# B&R Automation Studio project PLC code - cp (part 10)

#### PressureCtrl.st
```iecst
ACTION PressureCtrl:

	//Send the data from the configuration to the PID structure
	LoadPIDparam(ADR(pidParPressure), ADR(dataVacc.Parameters.parPID));

	xEnablePID := StatusCtrl=TRANSVAC_WAITING OR StatusCtrl=TRANSVAC_CONTROLLING;

	//**********************************************************************************
	// PID PID PID PID PID PID PID PID PID PID PID PID PID PID PID PID PID PID PID PID
	//**********************************************************************************
	fbPIDPressure.Enable:=xEnablePID;
	fbPIDPressure.PIDParameters:=pidParPressure;
	fbPIDPressure.MinOut:=0.0;
	fbPIDPressure.MaxOut:= dataVacc.Parameters.rMaxPIDOut;
	fbPIDPressure.Update:= xUpdatePID;
	fbPIDPressure.EnableTracking := StatusCtrl=TRANSVAC_WAITING; //This is the manual mode
	fbPIDPressure.TrackingValue := dataVacc.Parameters.rStartUpDutyCycle; //The StartUp value is defined as Manual
	fbPIDPressure.SetValue:=dataVacc.Parameters.rVacPressureSetPointPerc;
	fbPIDPressure.ActValue:=rVacPressurePerc;
	fbPIDPressure();

	//Assignation of the SetPoint of the Blower
	CASE StatusCtrl OF

		TRANSVAC_OFF:
			dataVacc.Status.Blower.rDutyCycle:=0.0;

		TRANSVAC_WAITING,
		TRANSVAC_CONTROLLING:
			dataVacc.Status.Blower.rDutyCycle:=MAX(dataVacc.Parameters.rMinDutyCycle, fbPIDPressure.Out);

		TRANSVAC_MAN:
			dataVacc.Status.Blower.rDutyCycle:=MAX(dataVacc.Parameters.rMinDutyCycle, dataVacc.parSw.rManSetPoint);

	END_CASE

	ValveControl;

END_ACTION

ACTION ValveControl:

	IF StatusCtrl = TRANSVAC_OFF OR NOT dataVacc.Parameters.Hw.xSystemWithJoints THEN
		//When machine is in 0 all valves should be open --> no vacuum
		dataVacc.Outputs.VacuumValves := 0;
	ELSE
		//When working, open the valves received from Sw in the command. If a Mask of minimum vaccum is desired, applied here
		dataVacc.Outputs.VacuumValves := NOT (dataVacc.parSw.ValvMask OR dataVacc.Parameters.MinValvMask) ;
	END_IF

	//Set the status the same as the physical outputs
	dataVacc.Status.VacuumValves := dataVacc.Outputs.VacuumValves;

END_ACTION
```

#### BlowerAlarms.st
```iecst
ACTION BlowerAlarms:

	//Comunication Alarm
	IF Blower.Status.ErrorComms THEN
		dataVacc.Alarms.xAlrComsBlower := TRUE;
		dataVacc.Alarms.xAlrCommsBlower[uiIndex] := TRUE;
	END_IF

	tonCheckAlarms.IN := dataVacc.Inputs.xSafetyEnable;
	tonCheckAlarms.PT := T#3000ms;
	tonCheckAlarms();

	//Driver Blower Error
	IF tonCheckAlarms.Q AND NOT dataVacc.Alarms.xAlrComsBlower AND
		((Blower.Status.ErrorID <> 0 AND Blower.Status.ErrorID <> 20625) OR Blower.Status.StatusErrorStop) THEN
			dataVacc.Alarms.xAlrDriveBlowerError := TRUE;
			dataVacc.Alarms.xAlrBlowerError[uiIndex] := TRUE;
	END_IF

	//Separate CB Blower Alarm
	IF tonCheckAlarms.Q AND NOT Blower.ElecSignals.In.xBreakerOK THEN
		dataVacc.Alarms.xAlrBlowerCB[uiIndex] := TRUE;
	END_IF

	IF FALSE THEN
		dataVacc.Alarms.xAlrOvertorque := TRUE;
	END_IF

	//Alarm if the blower has a speed configure higher than 0, has order to move and is stopped
	//Using Orders.PowerOn because Commands.MovePositive and Commands.MoveNegative are just edges
	tonBlowerNotRunning[uiIndex].IN := StatusCtrl <> TRANSVAC_OFF AND Blower.Parameters.Velocity > 40.0 AND ABS(Blower.Status.ActVelocity) < 40.0;
	tonBlowerNotRunning[uiIndex].PT := T#5s;
	tonBlowerNotRunning[uiIndex]();
	IF tonBlowerNotRunning[uiIndex].Q THEN
		dataVacc.Alarms.xAlrBlowerNotRunning[uiIndex] := TRUE;
	END_IF

END_ACTION
```

#### BlowerControl.st
```iecst
ACTION BlowerControl:

	IF NOT Blower.Status.StatusOperation THEN
		xAllBlowersRunning := FALSE;
	END_IF

	IF NOT Blower.Status.xAtSpeed THEN
		xAllBlowersAtSpeed := FALSE;
	END_IF

	//Define maximum DutyCycle if in Maximum mode
	IF StatusCtrl = TRANSVAC_MAXIMUM THEN
		dataVacc.Status.Blower.rDutyCycle := 100;
	END_IF

	//TODO: Need to change units. Order from PID in % and command in rpm
	Blower.Parameters.Velocity := REAL_TO_UINT(dataVacc.Status.Blower.rDutyCycle * dataVacc.Parameters.rMaxSpeed / 100);

	xEnteringPowerOn := NOT dataVacc.Parameters.Mode.xZero AND NOT Blower.Orders.PowerOn;
	Blower.Orders.PowerOn := NOT dataVacc.Parameters.Mode.xZero;

	ConditionStart := Blower.Status.ReadyForOrders AND StatusCtrl <> TRANSVAC_OFF;

	IF ConditionStart AND NOT ConditionStart_copy  THEN
		//TOREVIEW: Command should be an edge
		IF BlowerDirection = MOTOR_POSITIVE THEN
			Blower.Commands.MovePositive := TRUE;
		ELSIF BlowerDirection = MOTOR_NEGATIVE THEN
			Blower.Commands.MoveNegative := TRUE;
		END_IF
	END_IF

	IF StatusCtrl = TRANSVAC_OFF AND StatusCtrl_copy<> TRANSVAC_OFF THEN
		Blower.Commands.Stop := TRUE;
	END_IF

	IF dataVacc.Commands.xReset OR xEnteringPowerOn THEN
		Blower.Commands.Reset := TRUE;
	END_IF

END_ACTION
```

#### EventLog.st
```iecst
ACTION LogStopAlarm:

	stEventLog.Source := ELOG_TYPE_TRANS_VACUUM;
	stEventLog.Severity:= ELOG_SEVERITY_INFO;
	stEventLog.Facility:= iIndexTransVacuum;
	stEventLog.ErrorCode:=0;

	stEventLog.Text := 'Vacuum.LogStopAlarm';

	IF 		iReasonStop.0 THEN stEventLog.Text := 'Vacuum. xAlrVacuumSensor';
	ELSIF 	iReasonStop.1 THEN stEventLog.Text := 'Vacuum. xAlrComsBlower';
	ELSIF 	iReasonStop.2 THEN stEventLog.Text := 'Vacuum. xAlrDriveBlowerError';
	ELSIF 	iReasonStop.3 THEN stEventLog.Text := 'Vacuum. xAlrOvertorque';
	ELSIF 	iReasonStop.4 THEN stEventLog.Text := 'Vacuum. xAlrJointSystemPressure';
	ELSIF 	iReasonStop.5 THEN stEventLog.Text := 'Vacuum. xAlrBlowersAnyCB';
	ELSIF 	iReasonStop.6 THEN stEventLog.Text := 'Vacuum. xAlrBlowerCB[1]';
	ELSIF 	iReasonStop.7 THEN stEventLog.Text := 'Vacuum. xAlrBlowerCB[2]';
	END_IF

	gEventLogLoader(EventData := ADR(stEventLog));

END_ACTION
```

### Program Logical/ExtPack/_Transport/TransVacuumCtrl/TransVacuumSim/TransVacuumSim_v1/TransVacuumSim (IEC)

#### Main.st
```iecst
PROGRAM _INIT
	pressureSim.AnalogType := ANALOGSIM_EXPONENTIAL_POS;
	pressureSim.rInitialValue := 16384;
	//pressureSim.rNewPresentValue := 16384;
	pressureSim.rMinValue := 10900;
	pressureSim.rMaxValue := 16384;

	rAParam := 5;	//Fixed change
	rBParam := 0.010;	//Change with DC

END_PROGRAM

PROGRAM _CYCLIC

	transVacc ACCESS ADR(gTransVacuum[iTransVacummSimIndex]);

	pressureSim.rA := rAParam * transVacc.Parameters.rMaxSystemVacuum;
	pressureSim.rB := rBParam * transVacc.Parameters.rMaxSystemVacuum;

	pressureSim.rActionControl := transVacc.Status.Blower.rDutyCycle;
	//pressureSim.xUseNewValue := EDGEPOS(transVacc.Status.State<>TRANSVAC_OFF);
	pressureSim();
	transVacc.Inputs.iPressureRaw:=REAL_TO_INT(pressureSim.rPresentValue);

	tofNoVacc.IN := transVacc.Status.rVacPressure > 0.0;
	tofNoVacc.PT := t#100ms;
	tofNoVacc();
	transVacc.Inputs.xJointSystemPressure	:= tofNoVacc.Q;
	transVacc.Inputs.xVaccAirFlow	:= tofNoVacc.Q;

	//Increase the index for simulating the next item
	iTransVacummSimIndex := iTransVacummSimIndex +1;

END_PROGRAM
```

### JamDetect.typ
```iecst
TYPE
	JamVibrationStatus_enum :
		(
		JAMVIB_NOT_INSTALLED,
		JAMVIB_NOT_INIT,
		JAMVIB_TESTING,
		JAMVIB_WORKING,
		JAMVIB_WAITING
		);
	JamTestingStatus_enum :
		(
		JAMVIBT_INIT,
		JAMVIBT_ACTIVATE_SIGNAL,
		JAMVIBT_WAITING_TO_CHECK,
		JAMVIBT_CHECKING,
		JAMVIBT_GO_NEXT
		);
	JamDetectInputs_typ : 	STRUCT
		xJamCrash : ARRAY[0..4]OF BOOL; (*Crash Bar Signal*)
		xJamTestOk : BOOL; (*Jam detection test has failed signal*)
		xJamLowCrash : BOOL; (*Low level crash device signal*)
	END_STRUCT;
	JamDetectOutputs_typ : 	STRUCT
		xJamTestSignal : ARRAY[0..4]OF BOOL; (*Jam test output signal*)
	END_STRUCT;
	JamDetectAlarms_typ : 	STRUCT
		xAlrJamCrash : ARRAY[0..4]OF BOOL; (*Alarm Stop, Crash in bar has detected*)
		xAlrJamTest : ARRAY[0..4]OF BOOL; (*Alarm Stop, Test has failed*)
		xAlrJamLowCrash : BOOL; (*Alarm Warning, low level crash detected in unknow bar*)
	END_STRUCT;
	JamDetectParameters_typ : 	STRUCT
		xJamEnabled : BOOL; (*Jam detection has enabled*)
		iMappingJam : INT; (*Physical mapping of the JamDevice*)
		iBlock : USINT; (*Block where the JamDevice is installed*)
		iMappingBarPos : ARRAY[0..MAX_LAST_JAMSENSOR]OF USINT; (*Physical Mapping Bar Position of the sensor*)
		xBarInstalled : ARRAY[0..MAX_LAST_JAMSENSOR]OF BOOL; (*Bar Installed*)
		iSensorsQuantity : USINT; (*Number of bars controlled by module*)
		xDisableTest : BOOL; (*Disables the JAMVIB_TESTING step*)
		iLowJamTimes : ARRAY[0..1]OF USINT; (*Number of rise edges of xJamLowCrash to show alarm*)
		iLowJamCheckDuration : ARRAY[0..1]OF TIME; (*Period of time to check consecutive xJamLowCrash rise edges to show alarm*)
		xDisableLowJamAlarm : BOOL; (*Low level jam detection alarm disabled*)
	END_STRUCT;
	JamDetectCommands_typ : 	STRUCT
		xReset : BOOL; (*Reset signal*)
		xMuteAlarms : BOOL; (*Mute alarms signal*)
		xStart : BOOL; (*Do the test and check*)
		xPause : BOOL; (*Jam pause comand, belt stop, bars in print and block in auto*)
	END_STRUCT;
	JamDetect_typ : 	STRUCT
		Inputs : JamDetectInputs_typ;
		Outputs : JamDetectOutputs_typ;
		Alarms : JamDetectAlarms_typ;
		Status : JamVibrationStatus_enum;
		Parameters : JamDetectParameters_typ;
		Commands : JamDetectCommands_typ;
		AlSummary : stEFI_AlarmSummary;
	END_STRUCT;
	JamPerBar_typ : 	STRUCT
		iJamDevice : USINT;
		iJamSensor : USINT;
		xAlrJamCrash : BOOL;
		xAlrJamTest : BOOL;
		xAlrLowJamCrash : BOOL; (*Low level jam detection from jam device*)
	END_STRUCT;
END_TYPE
```

### JamDetect.var
```iecst
VAR
	iIndexJam : USINT;
END_VAR
```

- Program Logical/ExtPack/_Transport/JamDetectCtrl/JamDetect_v1/InitJamDetect (IEC) (no source held here)

### Program Logical/ExtPack/_Transport/JamDetectCtrl/JamDetect_v1/JamDetect (IEC)

#### JamDetect.st - Init, cyclic, exit code
```iecst
PROGRAM _CYCLIC

	JamDetect ACCESS ADR(gJamDetect[iIndexJam]);

	IF NOT JamDetect.Parameters.xJamEnabled THEN
		JamDetect.Alarms := AlarmsReseted;
		JamDetect.Commands := CommandsReseted;

		JamDetect.Status := JAMVIB_NOT_INSTALLED;
		xTestFinished := FALSE;

		iIndexJam := iIndexJam + 1;
		RETURN;
	END_IF

	(***RESET ALARMS***)
	IF JamDetect.Commands.xReset THEN
		JamDetect.Alarms := AlarmsReseted;
		JamDetect.AlSummary.xAlarmStop := FALSE;
	END_IF

	JamDetectCtrl;
	JamAlarmsSound;

	iIndexJam := iIndexJam + 1;

END_PROGRAM
```

#### JamDetectCtrl.st - Chiller control
```iecst
ACTION JamDetectCtrl:

	xStatusChanged := StatusPrevious <> JamDetect.Status ;
	StatusPrevious := JamDetect.Status;

	CASE JamDetect.Status OF
		JAMVIB_NOT_INSTALLED:
			JamDetect.Status := JAMVIB_NOT_INIT;

		JAMVIB_NOT_INIT:
			ResetTestingOrders;
			IF JamDetect.Commands.xStart THEN
				IF JamDetect.Parameters.xDisableTest THEN
					JamDetect.Status := JAMVIB_WORKING;
				ELSIF NOT xAnyTestAlarm THEN
					JamDetect.Status := JAMVIB_TESTING;
				END_IF
			END_IF

		JAMVIB_TESTING:

			JamTesting;

			IF xTestFinished THEN
				IF JamDetect.Commands.xStart AND NOT xAnyTestAlarm THEN
					xTestFinished := FALSE;
					JamDetect.Status := JAMVIB_WORKING;
				ELSE
					JamDetect.Status := JAMVIB_NOT_INIT;
				END_IF
			END_IF

		JAMVIB_WORKING:

			JamAlarms;

			IF JamDetect.Commands.xPause THEN
				JamDetect.Status := JAMVIB_WAITING;
			END_IF

			IF NOT JamDetect.Commands.xStart THEN
				JamDetect.Status := JAMVIB_NOT_INIT;
			END_IF

		JAMVIB_WAITING:

			IF NOT JamDetect.Commands.xPause THEN
				IF JamDetect.Commands.xStart THEN
					JamDetect.Status := JAMVIB_WORKING;
				ELSE
					JamDetect.Status := JAMVIB_NOT_INIT;
				END_IF
			END_IF

	END_CASE

	//Saving state history
	IF JamDetect.Status<>StateHistory[0] THEN
		FOR iIndexHistory:=iHistoryLines TO 1 BY -1 DO
			StateHistory[iIndexHistory]:=StateHistory[iIndexHistory-1];
		END_FOR;
		StateHistory[0]:=JamDetect.Status;
	END_IF

	//Alarm Summary
	xAnyCrashAlarm	:= FALSE;
	IF JamDetect.Status <> JAMVIB_TESTING THEN xAnyTestAlarm := FALSE; END_IF

	FOR iIndexSensor:=1 TO JamDetect.Parameters.iSensorsQuantity BY 1 DO
		IF JamDetect.Alarms.xAlrJamCrash[iIndexSensor] THEN xAnyCrashAlarm := TRUE; END_IF
		IF JamDetect.Alarms.xAlrJamTest[iIndexSensor] THEN	xAnyTestAlarm := TRUE; END_IF
	END_FOR
	JamDetect.AlSummary.xAlarmStop := xAnyCrashAlarm OR xAnyTestAlarm;

	JamDetect.AlSummary.xAnyWarning := JamDetect.Alarms.xAlrJamLowCrash;

END_ACTION
```

#### JamAlarms.st - Chiller control
```iecst
ACTION JamAlarms:

	(**CRASH ALARMS**)
	FOR iIndexSensor:=1 TO JamDetect.Parameters.iSensorsQuantity BY 1 DO
		//Jam Alarms if Enabled
		IF JamDetect.Parameters.xBarInstalled[iIndexSensor] THEN
			IF NOT JamDetect.Inputs.xJamCrash[iIndexSensor] THEN JamDetect.Alarms.xAlrJamCrash[iIndexSensor] := TRUE; END_IF
		END_IF
	END_FOR

	(** Low jam detection DELOREAN-2694 **)
	IF NOT JamDetect.Parameters.xDisableLowJamAlarm THEN
		tofConsecutiveLowJamDetected[0].IN := JamDetect.Inputs.xJamLowCrash;
		tofConsecutiveLowJamDetected[0].PT := JamDetect.Parameters.iLowJamCheckDuration[0];
		tofConsecutiveLowJamDetected[0]();

		ctuConsecutiveLowJamDetected[0].CU := JamDetect.Inputs.xJamLowCrash AND tofConsecutiveLowJamDetected[0].Q;
		ctuConsecutiveLowJamDetected[0].PV := JamDetect.Parameters.iLowJamTimes[0];
		ctuConsecutiveLowJamDetected[0].RESET := NOT tofConsecutiveLowJamDetected[0].Q;
		ctuConsecutiveLowJamDetected[0]();

		tofConsecutiveLowJamDetected[1].IN := JamDetect.Inputs.xJamLowCrash;
		tofConsecutiveLowJamDetected[1].PT := JamDetect.Parameters.iLowJamCheckDuration[1];
		tofConsecutiveLowJamDetected[1]();

		ctuConsecutiveLowJamDetected[1].CU := JamDetect.Inputs.xJamLowCrash AND tofConsecutiveLowJamDetected[1].Q;
		ctuConsecutiveLowJamDetected[1].PV := JamDetect.Parameters.iLowJamTimes[1];
		ctuConsecutiveLowJamDetected[1].RESET := NOT tofConsecutiveLowJamDetected[1].Q;
		ctuConsecutiveLowJamDetected[1]();

		IF ctuConsecutiveLowJamDetected[0].Q OR ctuConsecutiveLowJamDetected[1].Q THEN
			JamDetect.Alarms.xAlrJamLowCrash := TRUE;
			LogWarningAlarm;
		END_IF
	END_IF

END_ACTION
```

#### JamAlarmsSound.st
```iecst
ACTION JamAlarmsSound:

	//Auto reset sound management. All alarms need to work with mute option
	ars_AlrJamDetectionSound(xAlarm:=JamDetect.AlSummary.xAlarmStop, xSilence:=JamDetect.Commands.xMuteAlarms);

	//AutoReset alarms.

		JamDetect.AlSummary.xAlarmSound:=ars_AlrJamDetectionSound.xAlarmSound;

END_ACTION
```

### Program Logical/ExtPack/_Transport/JamDetectCtrl/JamDetectSim/JamDetectSim_v1/JamDetectSim (IEC)

#### Main.st - Init, cyclic, exit code
```iecst
PROGRAM _CYCLIC
	(* Insert code here *)

	JamDetectData  ACCESS ADR(gJamDetect[usiJamDetectSimIndex]);
	JamDataSim ACCESS ADR(gSimJamDetect[usiJamDetectSimIndex]);

	IF NOT JamDetectData.Parameters.xJamEnabled THEN
		usiJamDetectSimIndex := usiJamDetectSimIndex +1;
		RETURN;
	END_IF

	JamDetectData.Inputs.xJamCrash[1]:=JamDetectData.Parameters.xBarInstalled[1] AND NOT JamDataSim.Commands.CreateCrash[1];
	JamDetectData.Inputs.xJamCrash[2]:=JamDetectData.Parameters.xBarInstalled[2] AND NOT JamDataSim.Commands.CreateCrash[2];
	JamDetectData.Inputs.xJamCrash[3]:=JamDetectData.Parameters.xBarInstalled[3] AND NOT JamDataSim.Commands.CreateCrash[3];
	JamDetectData.Inputs.xJamCrash[4]:=JamDetectData.Parameters.xBarInstalled[4] AND NOT JamDataSim.Commands.CreateCrash[4];

	//Tests

	tonTestDelay.IN :=	(JamDetectData.Outputs.xJamTestSignal[1]  AND NOT JamDataSim.Commands.ErrorInTest[1]) OR
						(JamDetectData.Outputs.xJamTestSignal[2]  AND NOT JamDataSim.Commands.ErrorInTest[2]) OR
						(JamDetectData.Outputs.xJamTestSignal[3]  AND NOT JamDataSim.Commands.ErrorInTest[3]) OR
						(JamDetectData.Outputs.xJamTestSignal[4]  AND NOT JamDataSim.Commands.ErrorInTest[4]);
	tonTestDelay.PT := T#1s;
	tonTestDelay();
	JamDetectData.Inputs.xJamTestOk := tonTestDelay.Q;

	usiJamDetectSimIndex := usiJamDetectSimIndex + 1;

END_PROGRAM
```

#### JamDetectSim.var - Local variables
```iecst
VAR
	JamDetectData : REFERENCE TO JamDetect_typ;
	JamDataSim : REFERENCE TO JamDetectSim_typ;
	usiIndexTest : USINT;
	tonTestDelay : TON;
END_VAR
```

### JamDetectSim.typ
```iecst
TYPE
	JamDetectCommandsSim_typ : 	STRUCT
		ErrorInTest : ARRAY[0..4]OF BOOL;
		CreateCrash : ARRAY[0..4]OF BOOL;
	END_STRUCT;
	JamDetectSim_typ : 	STRUCT
		Commands : JamDetectCommandsSim_typ;
	END_STRUCT;
END_TYPE
```

### JamDetectSimGen.var
```iecst
VAR
	usiJamDetectSimIndex : USINT;
END_VAR
```

### EdgeHoldDown.typ
```iecst
TYPE
	EdgeHoldDown_typ : 	STRUCT
		ordersSw : EdgeHoldDownOrdersSw; (*Orders from sw*)
		commandsSw : EdgeHoldDownCommandsSw; (*Commands gui*)
		commands : EdgeHoldDownCommands; (*Commands gui*)
		orders : EdgeHoldDownOrders;
		parameters : EdgeHoldDownParameters; (*Parameters gui*)
		parSw : EdgeHoldDownParametersSw;
		status : EdgeHoldDownStatus; (*States potocell system*)
		Alarms : EdgeHoldDownAlarms; (*Alarms*)
		AlSummary : stEFI_AlarmSummary; (*Alarms Summary*)
		inputs : EdgeHoldDownInputs;
		Hw : EdgeHoldDownParametersHw_typ;
	END_STRUCT;
	EdgeHoldDownCommands : 	STRUCT
		xErrorRst : BOOL;
		xMute : BOOL;
		xStop : BOOL;
		AutoMode : stEFI_MachineAutoModes;
		Mode : StGeneral_States_Mode;
	END_STRUCT;
	EdgeHoldDownOrdersSw : 	STRUCT
		xMoveForward : BOOL;
		xMoveBackward : BOOL;
		xMoveUp : BOOL;
		xMoveDown : BOOL;
	END_STRUCT;
	EdgeHoldDownCommandsSw : 	STRUCT
		xReference : BOOL;
	END_STRUCT;
	EdgeHoldDownOrders : 	STRUCT
		xResetPosition : BOOL; (*Order to move adjustment systems to resting position*)
		xAdjustToMedia : BOOL; (*Order to move adjustment system to working position*)
	END_STRUCT;
	EdgeHoldDownParametersSw : 	STRUCT
		rBarsOffset : REAL := 15; (*Offset desired between metal bands height and bars position (mm)*)
		iOverlap : INT := 10; (*Overlap between metal bands and media (mm)*)
		xEnable : BOOL;
	END_STRUCT;
	EdgeHoldDownParameters : 	STRUCT
		xInstalled : BOOL; (*This variable is activated when this functionality is intalled and ready to be enabled*)
		xEnableMovements : BOOL; (*Movements are enabled. Safe to move the adjustment systems and not damage the bars*)
		rDistanceMetalBandToSki : REAL := 20; (*Distance between ski and metal band*)
		rWidthSp : REAL; (*Metal bands width position setpoint*)
		rBarsOffset : REAL; (*Offset desired between metal bands and printing bars height*)
		rBarsHeighSp : REAL; (*Bars heigh setpoint*)
		rBlockPosition : REAL; (*Block over ehd system position*)
		iAdjustmentSystemsNumber : USINT; (*Number of adjustment systems used by the edge hold down. Adjust system is composed by two motors*)
	END_STRUCT;
	EdgeHoldDownStatus : 	STRUCT
		xInstalled : BOOL;
		xEnabled : BOOL;
		xReferencing : BOOL;
		xReferenced : BOOL;
		xInRestingPosition : BOOL;
		xAdjustedToMedia : BOOL;
		xMoving : BOOL;
		xReady : BOOL;
		xInPosition : BOOL;
		iSystemState : EdgeHoldDownState := EHD_STOPPED;
		EdgeHoldDownType : EdgeHoldDownType_enum;
		rSkiPosition : REAL;
		xGoingRestPosition : BOOL;
		xAdjusting : BOOL;
		rBlockPrePrintingPosition : REAL := 40; (*Distance between ski and metal band*)
	END_STRUCT;
	EdgeHoldDownAlarms : 	STRUCT
		xParametersOutOfRange : BOOL; (*Active when order to adjust media received and parameters are out of requirements*)
		xMovementsNotEnabled : BOOL; (*Active when order to adjust to media received when movements are not enabled*)
		xJam : BOOL; (*Jam sensor has detect media while ehd is adjusted to media*)
		xNotReferenced : BOOL; (*System not referenced*)
	END_STRUCT;
	EdgeHoldDownState :
		(
		EHD_STOPPED,
		EHD_MANUAL,
		EHD_IDLE,
		EHD_ERROR
		);
	EdgeHoldDownAutoState :
		(
		EHD_OUT_OF_AUTO,
		EHD_MOVEMENTS_NOT_ENABLED,
		EHD_READY,
		EHD_ADJUSTING_STEP_1,
		EHD_ADJUSTING_STEP_2,
		EHD_ADJUSTING_STEP_3,
		EHD_RESTING_STEP_1,
		EHD_RESTING_STEP_2,
		EHD_RESTING_STEP_3
		);
	EdgeHoldDownPositionStates :
		(
		UNDEFINED,
		HOMING,
		RESTING_POSITION,
		GOING_TO_WORKING_POSITION,
		WORKING_POSITION,
		GOING_TO_RESTING_POSITION
		);
	EdgeHoldDownOutputs : 	STRUCT
	END_STRUCT;
	EdgeHoldDownInputs : 	STRUCT
		xJam : BOOL;
	END_STRUCT;
	EdgeHoldDownType_enum :
		(
		EHDTY_UNDEFINED,
		EHDTY_V1,
		EHDTY_V2
		);
	EdgeHoldDownParametersHw_typ : 	STRUCT
		iMinBarsOffset : UINT := 10;
		iMaxBarsOffset : UINT := 15;
		iMinOverlap : INT := 8;
		iMaxOverlap : INT := 15;
		rMinWidthAdjustment : REAL := 424; (*Distance between sliders when inductive sensor for minimum position is active*)
		rMaxDistanceMetalBandToBelt : REAL := 60; (*Limited height where ehd can be moved vertically when postioned wider than belt's widht to avoid crash with 6l chassis*)
	END_STRUCT;
END_TYPE
```

- EdgeHoldDown.graphml (not shown)

### Program Logical/ExtPack/_Transport/EdgeHoldDown/EdgeHoldDown_v1/EdgeHoldDown (IEC)

#### EdgeHoldDown.st - Init, cyclic, exit code
```iecst
PROGRAM _INIT
	FOR iIndexHistory:=0 TO iHistoryLines DO
		StateHistory[iIndexHistory]:=EHD_STOPPED;
	END_FOR
END_PROGRAM

PROGRAM _CYCLIC

	//////////////////////////////
	////// ASSIGN LOCAL VARS //////
	//////////////////////////////

	//Main data assignation
	data ACCESS ADR (gEdgeHoldDown);
	AdjustmentSystem ACCESS ADR (gPairedMotors);

	data.status.xInstalled := data.parameters.xInstalled;

	IF EDGEPOS(data.parSw.xEnable) THEN
		data.status.xEnabled:=TRUE;

	//EHD may be disabled whether is positioned over the belt guide (Resting position)
	ELSIF ((NOT data.parSw.xEnable AND data.commands.Mode.xAuto) OR EDGEPOS(NOT data.parSw.xEnable)) AND data.status.xInRestingPosition THEN
		data.status.xEnabled := FALSE;
	END_IF

	Configuration;

	data.parameters.iAdjustmentSystemsNumber := LIMIT(1, data.parameters.iAdjustmentSystemsNumber, MAX_EHD_ADJUST_SYSTEMS);
	data.parameters.xEnableMovements := ((AdjustmentSystem[1].Motor[1].rPositionMotor + iSafetyOffset) < data.parameters.rBlockPosition); //Review how to set this condition when more than one block is installed

	IF NOT data.status.xInstalled OR NOT data.status.xEnabled THEN
		data.Alarms:= stAlarmsReseted;
		data.AlSummary := stEhdAlarmSummaryReseted;
		data.AlSummary.xAlarmSound:=FALSE;

		data.status.iSystemState:= EHD_STOPPED;
		data.status.xReferenced:=FALSE;
		ResetSwOrders;
		RETURN;
	END_IF

	//Reset alarms
	IF data.commands.xErrorRst THEN data.Alarms:= stAlarmsReseted; END_IF

	//States manager
	MachineState;

	//Alarms
	AlarmsSummary;

	///////////////////////
	//Alarm Sound
	AlarmSounds;

	//Resetting commands coming from sw
	data.commandsSw := ResetCommandsSw;

END_PROGRAM
```

#### AlarmsSummary.st - alarms summary
```iecst
ACTION AlarmsSummary:

	//////////////////////////
	////// RESET ALARMS //////
	//////////////////////////
	// Pending do commands gdata.commands.xReset
	IF data.commands.xErrorRst THEN
		data.Alarms := stAlarmsReseted;
		data.AlSummary := stEhdAlarmSummaryReseted;
	END_IF

	//Alarms
	IF data.status.xMoving AND NOT data.parameters.xEnableMovements THEN
		data.Alarms.xMovementsNotEnabled:=TRUE;
	END_IF

	IF data.status.xAdjustedToMedia AND data.inputs.xJam THEN
		data.Alarms.xJam:=TRUE;
	END_IF

	IF data.orders.xAdjustToMedia THEN
		IF ((AdjustmentSystem[1].parameters.rMechPositionMax + 2) < AdjustmentSystem[1].parameters.rPositionDesired) OR
			((AdjustmentSystem[1].parameters.rMechPositionMin - 2) > AdjustmentSystem[1].parameters.rPositionDesired) OR
			((AdjustmentSystem[2].parameters.rMechPositionMax + 2) < AdjustmentSystem[2].parameters.rPositionDesired) OR
			((AdjustmentSystem[2].parameters.rMechPositionMin - 2) > AdjustmentSystem[2].parameters.rPositionDesired) THEN

			data.Alarms.xParametersOutOfRange:=TRUE;
		END_IF
	END_IF

	//Alarms summary
	//Stop
	iReasonStop.0 := AdjustmentSystem[1].AlSummary.xAlarmStop;
	iReasonStop.1 := AdjustmentSystem[2].AlSummary.xAlarmStop;
	iReasonStop.2 := data.Alarms.xNotReferenced;
	iReasonStop.3 := data.Alarms.xParametersOutOfRange;

	data.AlSummary.xAlarmStop := iReasonStop > 0;
	IF EDGEPOS(data.AlSummary.xAlarmStop) THEN
		data.AlSummary.iReasonStop[0] := iReasonStop;
		LogStopAlarm;
	ELSIF EDGEPOS(NOT data.commands.AutoMode.xStop AND NOT data.AlSummary.xAlarmStop) THEN
		data.AlSummary.iReasonStop[0] := 0;
	END_IF

	//Critical
	iReasonCritical.0 := AdjustmentSystem[1].AlSummary.xAlarmCritical;
	iReasonCritical.1 := AdjustmentSystem[2].AlSummary.xAlarmCritical;
	iReasonCritical.2 := data.Alarms.xMovementsNotEnabled;
	iReasonCritical.3 := data.Alarms.xJam;

	data.AlSummary.xAlarmCritical := iReasonCritical > 0;
	IF EDGEPOS(data.AlSummary.xAlarmCritical) THEN
		data.AlSummary.iReasonCritical := iReasonCritical;
		LogCriticalAlarm;
	ELSIF EDGEPOS(data.commands.Mode.xAuto AND NOT data.AlSummary.xAlarmCritical) THEN
		data.AlSummary.iReasonCritical := 0;
	END_IF

	//Warning
	// It is just used for drive alarms
	iAnyWarning.0 := AdjustmentSystem[1].AlSummary.xAnyWarning;
	iAnyWarning.1 := AdjustmentSystem[2].AlSummary.xAnyWarning;

	data.AlSummary.xAnyWarning:= iAnyWarning > 0;
	IF EDGEPOS(data.AlSummary.xAnyWarning) THEN
		data.AlSummary.iReasonWarning := iAnyWarning;
		LogWarningAlarm;
	ELSIF EDGEPOS(NOT data.AlSummary.xAnyWarning) THEN
		data.AlSummary.iReasonWarning := 0;
	END_IF

END_ACTION
```

#### AlarmSounds.st
```iecst
ACTION AlarmSounds:

	// Alarms reseteable sound management.
	ars_AlrStop.xAlarm:= data.AlSummary.xAlarmStop;
	ars_AlrStop.xSilence:= data.commands.xMute;
	ars_AlrStop();

	ars_AlrCritical.xAlarm:= data.AlSummary.xAlarmCritical;
	ars_AlrCritical.xSilence:= data.commands.xMute;
	ars_AlrCritical();

	ars_AlrWarning.xAlarm:= data.AlSummary.xAnyWarning;
	ars_AlrWarning.xSilence:= data.commands.xMute;
	ars_AlrWarning();

	data.AlSummary.xAlarmSound:= //ars_AlrWarning.xAlarmSound OR
									ars_AlrStop.xAlarmSound OR
									ars_AlrCritical.xAlarmSound;

END_ACTION
```

#### EventLog.st
```iecst
ACTION LogWarningAlarm:

	stWarningAlarmsLog.Source := ELOG_TYPE_EHD;
	stWarningAlarmsLog.Severity:= ELOG_SEVERITY_INFO;
	stWarningAlarmsLog.Facility:= 0;
	stWarningAlarmsLog.ErrorCode:=0;

	stWarningAlarmsLog.Text := 'EHD.LogWarningAlarm';

	IF iReasonWarning.0 THEN stWarningAlarmsLog.Text := 'AdjustmentSystem[1].AlSummary.xAnyWarning';
	ELSIF iReasonWarning.1 THEN	stWarningAlarmsLog.Text := 'AdjustmentSystem[2].AlSummary.xAnyWarning';
	END_IF

	gEventLogLoader(EventData := ADR(stWarningAlarmsLog));

END_ACTION

ACTION LogStopAlarm:

	stStopAlarmsLog.Source := ELOG_TYPE_EHD;
	stStopAlarmsLog.Severity:= ELOG_SEVERITY_INFO;
	stStopAlarmsLog.Facility:= 0;
	stStopAlarmsLog.ErrorCode:=0;

	stStopAlarmsLog.Text := 'EHD.LogStopAlarm';

	IF iReasonStop.0 THEN stStopAlarmsLog.Text := 'AdjustmentSystem[1].AlSummary.xAlarmStop';
	ELSIF iReasonStop.1 THEN stStopAlarmsLog.Text := 'AdjustmentSystem[2].AlSummary.xAlarmStop';
	ELSIF iReasonStop.2 THEN stStopAlarmsLog.Text := 'data.Alarms.xNotReferenced';
	ELSIF iReasonStop.3 THEN stStopAlarmsLog.Text := 'data.Alarms.xParametersOutOfRange';
	END_IF

	gEventLogLoader(EventData := ADR(stStopAlarmsLog));

END_ACTION

ACTION LogCriticalAlarm:

	stCriticalAlarmsLog.Source := ELOG_TYPE_EHD;
	stCriticalAlarmsLog.Severity:= ELOG_SEVERITY_ERROR;
	stCriticalAlarmsLog.Facility:= 0;
	stCriticalAlarmsLog.ErrorCode:=0;

	stWarningAlarmsLog.Text := 'EHD.LogCriticalAlarm';

	IF iReasonCritical.0 THEN stWarningAlarmsLog.Text := 'AdjustmentSystem[1].AlSummary.xAlarmCritical';
	ELSIF iReasonCritical.1 THEN stWarningAlarmsLog.Text := 'AdjustmentSystem[2].AlSummary.xAlarmCritical';
	ELSIF iReasonCritical.2 THEN stWarningAlarmsLog.Text := 'data.Alarms.xMovementsNotEnabled';
	ELSIF iReasonCritical.3 THEN stWarningAlarmsLog.Text := 'data.Alarms.xJam';
	END_IF

	gEventLogLoader(EventData := ADR(stCriticalAlarmsLog));

END_ACTION
```

- Program Logical/ExtPack/_Transport/PairedIclaMotors/PairedIclaMotors_v1/InitPairedIclaMotors (IEC) (no source held here)

### Program Logical/ExtPack/_Transport/PairedIclaMotors/PairedIclaMotors_v1/PairedIclaMotors (IEC)

#### PairedIclaMotors.st - Init, cyclic, exit code
```iecst
PROGRAM _INIT
	FOR iIndexHistory:=0 TO iHistoryLines DO
		StateHistory[iIndexHistory]:=NOT_USED;
	END_FOR
END_PROGRAM

PROGRAM _CYCLIC

	//Main data assignation
	data ACCESS ADR (gPairedMotors[iIndexPairedIclaMotors]);
	IclaMaster ACCESS ADR (gIcla[gPairedMotors[iIndexPairedIclaMotors].parameters.IndexIclaMaster]);
	IclaGear ACCESS ADR (gIcla[gPairedMotors[iIndexPairedIclaMotors].parameters.IndexIclaGear]);

	IndexIclaMaster:=gPairedMotors[iIndexPairedIclaMotors].parameters.IndexIclaMaster;
	IndexIclaGear:=gPairedMotors[iIndexPairedIclaMotors].parameters.IndexIclaGear;

	//Review limits
	iNumIclaMotors := LIMIT(1, data.parameters.iNumIclaMotors, MAX_EHD_MOTORS_PER_ADJUST_SYS);
	rPositionDesired := LIMIT(data.parameters.rMechPositionMin, data.parameters.rPositionDesired, data.parameters.rMechPositionMax);

	data.status.xInstalled := data.parameters.xInstalled;
	IF data.status.xInstalled THEN
		//Motors data
		FOR iIndexIclaMotor:=1 TO iNumIclaMotors DO
			//Motor parameters
			dataToMotors;
			dataFromMotors;

			//Conversions
			IF data.parameters.xPositionSensorInstalled THEN
				Conversions;
			END_IF
		END_FOR
	END_IF

	data.status.xEnabled := data.parameters.xEnabled;
	IF NOT data.status.xEnabled THEN

		data.Alarms:= stAlarmsReseted;
		data.AlSummary := stAlarmSummaryReseted;
		data.AlSummary.xAlarmSound:=FALSE;

		data.status.xReferenced:=FALSE;
		ResetCommands;

		//Prepare for the next element
		iIndexPairedIclaMotors:= iIndexPairedIclaMotors +1;

		RETURN;
	END_IF

	IclaMotors[1]:=IclaMaster;
	IclaMotors[2]:=IclaGear;

	//Resetting commands
	IF data.commands.Mode.xZero THEN
		ResetCommands;
	END_IF

	//Motors state
	MotorsMachineState;

	// ALARMS
	AlarmsSummary;

	//Alarm Sound
	AlarmSounds;

	//Assigning motor data
	IclaMaster := IclaMotors[1];
	IclaGear := IclaMotors[2];

	//Prepare for the next element
	iIndexPairedIclaMotors:= iIndexPairedIclaMotors +1;

END_PROGRAM
```

#### MotorsMachineState.st - states control
```iecst
ACTION MotorsMachineState:

	xManualMovementEnabled := 	(iSystemState=MANUAL) OR
								(iSystemState=JOGGING) OR
								(iSystemState=HOMING_STEP_1) OR
								(iSystemState=HOMING_STEP_2) OR
								(iSystemState=HOMING_STEP_3);

	//Check motors are positioned in desired position
	IF (iSystemState=MANUAL) OR (iSystemState=JOGGING) THEN
		AssignJogOrders;
	END_IF
	CheckAnyManualMovement;
	CheckAnyManualOrder;

	CheckMotorStopped;
	//CheckMotorReferenced;
	CheckMotorReady;
	CheckMotorPositioned;

	CASE iSystemState OF

		NOT_INITIALIZED:
			ResetMotorsCommands;
			RemoveOrderMoveAbsolute;

			IF NOT xMotorStopped THEN
				SetStopOrder;
			ELSE
				CheckControllerReady;
				IF xControllerReady THEN
					iSystemState:=POWER_ON;
				END_IF
			END_IF

		POWER_ON:
			RemoveStopOrder;
			SetPowerOn;
			CheckPowerOn;
			IF xPoweredOn THEN
				//Go directly to wait homing process
				iSystemState:=POWERED;
			END_IF

		POWERED:
			IF xMotorReady THEN
				iSystemState := STANDSTILL;
			END_IF

		STANDSTILL:
			IF data.commands.Mode.xManual THEN
				iSystemState:=MANUAL;

			ELSIF data.commands.Mode.xAuto AND xMotorsReferenced AND data.parameters.xMovementsEnabled THEN
				iSystemState := AUTO;
			END_IF

		MANUAL:
			IF EDGEPOS(data.commands.xReference) THEN
				xMotorsReferenced := FALSE;
				iSystemState := HOMING_STEP_1;

			ELSIF xAnyManualMovement THEN
				iSystemState:=JOGGING;
			END_IF

		JOGGING:
			CheckMotorReady;
			IF NOT xAnyManualOrder THEN
				iSystemState := STANDSTILL;
			END_IF

		HOMING_STEP_1:
			//To home directly if both homing sensors are active
			CheckReferencePositionReached;
			IF xReferencePositionReached AND xMotorReady THEN
				iSystemState := HOMING_STEP_2;
			END_IF

		HOMING_STEP_2:
			//Execute home order
			SetHomeOrder;
			IF xMotorReady THEN
				iSystemState := HOMING_STEP_3;
			END_IF

		HOMING_STEP_3:
			CheckMotorReferenced;
			IF xMotorsReferenced THEN
				iSystemState := STANDSTILL;
			ELSE
				RemoveHomeOrder;
				iSystemState := HOMING_STEP_2;
			END_IF

		AUTO:
			RemoveStopOrder;
			IF xMotorReady THEN
				IF NOT xMotorsInPosition THEN
					SetOrderMoveAbsolute;
				END_IF
			ELSE
				iSystemState := NOT_INITIALIZED;
			END_IF

			IF data.status.xMoving THEN
				iSystemState := RUNNING;
			END_IF

		RUNNING:
			//If the movement is finished or the desired position has changed
			tonMotorStopped(IN:=xMotorStopped, PT:=T#500ms);
			IF xMotorsInPosition OR tonMotorStopped.Q OR data.commands.xStop THEN
				RemoveOrderMoveAbsolute;
				SetStopOrder;
				iSystemState := AUTO;
			END_IF

		ERROR:
			ResetMotorsCommands;
			//SetPowerOff;
			RemoveOrderMoveAbsolute;
			IF NOT xMotorStopped THEN
				SetStopOrder;
			END_IF

			IF NOT xAnyMotorError THEN
				iSystemState:=NOT_INITIALIZED;
			END_IF
	END_CASE

	//To check motors errors
	CheckAnyError;

	IF NOT data.parameters.xMovementsEnabled AND ((iSystemState = RUNNING) OR (iSystemState = AUTO)) THEN
		RemoveOrderMoveAbsolute;
		iSystemState := STANDSTILL;
	END_IF

	//Sending to ERROR
	IF xAnyMotorError OR data.AlSummary.xAlarmCritical THEN
		iSystemState:=ERROR;
	END_IF

	//In Zero mode it goes to not Init
	IF (data.commands.Mode.xZero) THEN
		iSystemState:=NOT_INITIALIZED;
	END_IF

	//Saving state history
	IF iSystemState<>StateHistory[0] THEN
		FOR iIndexHistory:=iHistoryLines TO 1 BY -1 DO
			StateHistory[iIndexHistory]:=StateHistory[iIndexHistory-1];
		END_FOR
		StateHistory[0]:=iSystemState;
	END_IF

	//State summary
	data.status.xInPosition := xMotorsInPosition;
	data.status.xMoving := NOT xMotorStopped;
	data.status.xReferenced	:= xMotorsReferenced;
	data.status.xReferencing :=	(iSystemState=HOMING_STEP_1) OR (iSystemState=HOMING_STEP_2) OR (iSystemState=HOMING_STEP_3);
	data.status.iSystemState := iSystemState;

END_ACTION

ACTION ResetMotorsCommands:
	FOR iIndexIclaMotor:=1 TO iNumIclaMotors DO
		IclaMotors[iIndexIclaMotor].Command.Enable := FALSE;
		IclaMotors[iIndexIclaMotor].Command.JogBackward := FALSE;
		IclaMotors[iIndexIclaMotor].Command.JogForward := FALSE;
		IclaMotors[iIndexIclaMotor].Command.MoveAbsolute := FALSE;
	END_FOR
END_ACTION

ACTION CheckControllerReady:
	xControllerReady:=TRUE;
	FOR iIndexIclaMotor:=1 TO iNumIclaMotors DO
		IF IclaMotors[iIndexIclaMotor].Status.Error.Communication THEN
			xControllerReady:=FALSE;
		END_IF
	END_FOR
END_ACTION

ACTION SetPowerOn:
	FOR iIndexIclaMotor:=1 TO iNumIclaMotors DO
		IclaMotors[iIndexIclaMotor].Command.Enable := TRUE;
	END_FOR
END_ACTION

ACTION SetPowerOff:
	FOR iIndexIclaMotor:=1 TO iNumIclaMotors DO
		IclaMotors[iIndexIclaMotor].Command.Enable := FALSE;
	END_FOR
END_ACTION

ACTION CheckPowerOn:
	xPoweredOn:=TRUE;
	FOR iIndexIclaMotor:=1 TO iNumIclaMotors DO
		IF (IclaMotors[iIndexIclaMotor].Status.IclaStatus<>AXISILE_POWER) AND (IclaMotors[iIndexIclaMotor].Status.IclaStatus<>AXISILE_READY) THEN
			xPoweredOn:=FALSE;
		END_IF
	END_FOR
END_ACTION

ACTION CheckMotorReady:
	xMotorReady:=TRUE;
	FOR iIndexIclaMotor:=1 TO iNumIclaMotors DO
		IF (IclaMotors[iIndexIclaMotor].Status.iDriveStatus<>ICLAST_ENABLE_OPERATION) THEN
			xMotorReady:=FALSE;
		END_IF
	END_FOR
END_ACTION

ACTION SetHomeOrder:
	FOR iIndexIclaMotor:=1 TO iNumIclaMotors DO
		IF IclaMotors[iIndexIclaMotor].Status.iActualVelocity = 0 THEN
			IclaMotors[iIndexIclaMotor].Command.Home := TRUE;
		END_IF
	END_FOR
END_ACTION

ACTION RemoveHomeOrder:
	FOR iIndexIclaMotor:=1 TO iNumIclaMotors DO
		IclaMotors[iIndexIclaMotor].Command.Home := FALSE;
	END_FOR
END_ACTION

ACTION SetOrderGoingForward:
	data.commands.xMoveForward := TRUE;
END_ACTION

ACTION RemoveOrderGoingForward:
	data.commands.xMoveForward := FALSE;
END_ACTION

ACTION SetOrderGoingBackward:
	data.commands.xMoveBackward := TRUE;
END_ACTION

ACTION RemoveOrderGoingBackward:
	data.commands.xMoveBackward := FALSE;
END_ACTION

ACTION SetOrderMoveAbsolute:
	rCopyPositionDesired := rPositionDesired;
	FOR iIndexIclaMotor:=1 TO iNumIclaMotors DO
		MotorDriveUnit.PositionDesired := data.Motor[iIndexIclaMotor].iDirection * rPositionDesired;
		MotorDriveUnit.Calculation := CALC_POS_PULSES;
		MotorDriveUnit();

		IclaMotors[iIndexIclaMotor].Parameter.MoveAbsolute.Position := REAL_TO_DINT(MotorDriveUnit.pulsesPositionDesired);
		IclaMotors[iIndexIclaMotor].Command.MoveAbsolute := TRUE;
	END_FOR
END_ACTION

ACTION RemoveOrderMoveAbsolute:
	FOR iIndexIclaMotor:=1 TO iNumIclaMotors DO
		IclaMotors[iIndexIclaMotor].Command.MoveAbsolute := FALSE;
	END_FOR
END_ACTION

ACTION SetStopOrder:
	FOR iIndexIclaMotor:=1 TO iNumIclaMotors DO
		IclaMotors[iIndexIclaMotor].Command.Stop := TRUE;
	END_FOR
END_ACTION

ACTION RemoveStopOrder:
	FOR iIndexIclaMotor:=1 TO iNumIclaMotors DO
		IclaMotors[iIndexIclaMotor].Command.Stop := FALSE;
	END_FOR
END_ACTION

ACTION AssignJogOrders:
	FOR iIndexIclaMotor:=1 TO iNumIclaMotors DO
		//[RGP] Ehd width fitting exit motor direction is not the same as the one on the entry side due to mechanical assembly.
		//This case does not apply to elevation motors, which are mechanically assembled the same way.
		IF iIndexPairedIclaMotors=2 AND iIndexIclaMotor=2 THEN
			IclaMotors[iIndexIclaMotor].Command.JogBackward := data.commands.xMoveForward AND NOT data.commands.xMoveBackward AND NOT data.Motor[iIndexIclaMotor].Inputs.xMinPositionReached;
			IclaMotors[iIndexIclaMotor].Command.JogForward := data.commands.xMoveBackward AND NOT data.commands.xMoveForward AND NOT data.Motor[iIndexIclaMotor].Inputs.xMaxPositionReached;
		ELSE
			IclaMotors[iIndexIclaMotor].Command.JogForward := data.commands.xMoveForward AND NOT data.commands.xMoveBackward AND NOT data.Motor[iIndexIclaMotor].Inputs.xMinPositionReached;
			IclaMotors[iIndexIclaMotor].Command.JogBackward := data.commands.xMoveBackward AND NOT data.commands.xMoveForward AND NOT data.Motor[iIndexIclaMotor].Inputs.xMaxPositionReached;
		END_IF
	END_FOR
END_ACTION

ACTION CheckAnyManualOrder:
	xAnyManualOrder := 	IclaMotors[1].Command.JogForward OR
						IclaMotors[1].Command.JogBackward OR
						IclaMotors[2].Command.JogForward OR
						IclaMotors[2].Command.JogBackward;
END_ACTION

ACTION CheckAnyManualMovement:
	xAnyManualMovement := FALSE;
	FOR iIndexIclaMotor:=1 TO iNumIclaMotors DO
		IF (IclaMotors[iIndexIclaMotor].Status.IclaStatus = AXISILE_JOG) THEN
			xAnyManualMovement := TRUE;
		END_IF
	END_FOR
END_ACTION

ACTION CheckAnyError:
	xAnyMotorError:=FALSE;
	FOR iIndexIclaMotor:=1 TO iNumIclaMotors DO
		// Not comms
		data.Motor[iIndexIclaMotor].Alarms.xCommsMotorError := FALSE;
		IF (IclaMotors[iIndexIclaMotor].Status.Error.Communication) THEN
			data.Motor[iIndexIclaMotor].Alarms.xCommsMotorError := TRUE;
		END_IF

		// Motor Error
		data.Motor[iIndexIclaMotor].Alarms.xMotorError := FALSE;
		IF ((IclaMotors[iIndexIclaMotor].Status.iDriveStatus = ICLAST_ERROR) OR
			IclaMotors[iIndexIclaMotor].Status.Error.ErrorNumber<>0) THEN
			data.Motor[iIndexIclaMotor].Alarms.xMotorError := TRUE;
		END_IF

		// Motor Error
		data.Motor[iIndexIclaMotor].Alarms.xControllerNotReady := FALSE;
		IF (IclaMotors[iIndexIclaMotor].Status.iDriveStatus = ICLAST_SWITCH_ON_DISABLED) THEN
			data.Motor[iIndexIclaMotor].Alarms.xControllerNotReady := TRUE;
		END_IF

	END_FOR
END_ACTION

ACTION CheckMotorStopped:
	xMotorStopped := TRUE;
	FOR iIndexIclaMotor:=1 TO iNumIclaMotors DO
		IF (IclaMotors[iIndexIclaMotor].Status.iActualVelocity <> 0) THEN
			xMotorStopped:=FALSE;
		END_IF
	END_FOR
END_ACTION

ACTION CheckReferencePositionReached:
	IF iIndexPairedIclaMotors=1 THEN
		//Elevation motors
		xReferencePositionReached := data.Motor[1].Inputs.xMinPositionReached AND data.Motor[2].Inputs.xMinPositionReached;
	ELSE
		//Width fitting motors
		xReferencePositionReached := data.Motor[1].Inputs.xMaxPositionReached AND data.Motor[2].Inputs.xMaxPositionReached;
	END_IF
END_ACTION

ACTION CheckMotorPositioned:
	xMotorsInPosition := TRUE;
	FOR iIndexIclaMotor:=1 TO iNumIclaMotors DO
		IF (ABS(data.Motor[iIndexIclaMotor].rPositionMotor - rPositionDesired) > data.Motor[iIndexIclaMotor].rMotorResolution) THEN
			xMotorsInPosition := FALSE;
		END_IF
	END_FOR
END_ACTION

ACTION CheckMotorReferenced:
	xMotorsReferenced := TRUE;
	FOR iIndexIclaMotor:=1 TO iNumIclaMotors DO
		IF NOT IclaMotors[iIndexIclaMotor].Status.xReferenced THEN
			xMotorsReferenced := FALSE;
		ELSE
			//Distance between sensors calculated instead of being a hardware defined parameter. Just for testing, this parameters must be defined by mechanical team
			data.Motor[iIndexIclaMotor].rDistanceBetweenSensors := (ABS(data.Motor[iIndexIclaMotor].rHomePosition)*2 + gEdgeHoldDown.Hw.rMinWidthAdjustment) - (data.Motor[iIndexIclaMotor].rMeasuredPositionFrontSide + data.Motor[iIndexIclaMotor].rMeasuredPositionBackSide);
		END_IF
	END_FOR
END_ACTION
```

#### Conversions.st
```iecst
ACTION Conversions:

	//There are two distance sensor per motor

	//y = mx + b
	//y = distance measured (mm)
	//x = value read by sensor
	//b = value of distance at minimum analogic value read (4mA) = 100mm
	//sensor maximum measure distance is 600

	//y(x)=0.0183x + 58 //Practical. (RawUnits)

	//Front sensor
	data.Motor[iIndexIclaMotor].rMeasuredPositionFrontSide := (data.Motor[iIndexIclaMotor].Inputs.iMeasuredPositionFrontSide*rSlopeAnalogSensor + rInterceptAnalogSensor);

	//Back sensor
	data.Motor[iIndexIclaMotor].rMeasuredPositionBackSide := (data.Motor[iIndexIclaMotor].Inputs.iMeasuredPositionBackSide*rSlopeAnalogSensor + rInterceptAnalogSensor);

	//Distance between metal bands/straps
	rMeasuredDistanceMetalStraps[iIndexIclaMotor] := 	data.Motor[iIndexIclaMotor].rMeasuredPositionFrontSide +
														data.Motor[iIndexIclaMotor].rMeasuredPositionBackSide +
														data.Motor[iIndexIclaMotor].rDistanceBetweenSensors;

	IF ABS(data.Motor[iIndexIclaMotor].rMeasuredDistanceMetalStraps - rMeasuredDistanceMetalStraps[iIndexIclaMotor])> rAnalogSensorTolerance THEN
		data.Motor[iIndexIclaMotor].rMeasuredDistanceMetalStraps := rMeasuredDistanceMetalStraps[iIndexIclaMotor];
	END_IF

END_ACTION
```

#### AlarmsSummary.st - alarms summary
```iecst
ACTION AlarmsSummary:

	//RESET ALARMS
	IF data.commands.xErrorRst THEN
		data.Alarms := stAlarmsReseted;
		data.AlSummary := stAlarmSummaryReseted;
	END_IF

	//Invalid position
	IF data.status.xReferenced AND data.status.xMoving THEN
		IF (rPositionMotorMm > (data.parameters.rMechPositionMax + data.Motor[1].rMotorResolution)) OR ((rPositionMotorMm < data.parameters.rMechPositionMin - data.Motor[1].rMotorResolution)) THEN
			data.Alarms.xPositionOutOfRange := TRUE;
		END_IF
	END_IF

	//Alarm Not referenced
	data.Alarms.xNotReferenced:= NOT data.status.xReferenced;

	//////////////////////////////////////////
	//To review in next releases how to share with SW an alarm per motor and not per adjustment system. To improve troubleshooting

	//Error general. Check error id for more information
	data.Alarms.xMotorError:=data.Motor[1].Alarms.xMotorError OR data.Motor[2].Alarms.xMotorError;

	//Enables (STO)
	IF data.Inputs.xSafetyEnable AND NOT data.commands.Mode.xZero THEN
		data.Alarms.xControllerNotReady :=  data.Motor[1].Alarms.xControllerNotReady OR data.Motor[2].Alarms.xControllerNotReady;
	END_IF

	//Comms
	data.Alarms.xCommsMotorError:=data.Motor[1].Alarms.xCommsMotorError OR data.Motor[2].Alarms.xCommsMotorError;

	xAnyMotorError := data.Alarms.xMotorError OR data.Alarms.xCommsMotorError;

	//////////////////////////////////////////

	//Motors not aligned
	data.Alarms.xNotAligned := ABS(data.Motor[1].rPositionMotor-data.Motor[2].rPositionMotor) > data.parameters.iMisalignmentTolerance;

	//Inconsistency between position measured (analogic input) and motor position information (motors encoder)
	iPositionMeasuredInconsistency.0 := ABS(data.Motor[1].rMetalStrapPos-data.Motor[1].rMeasuredDistanceMetalStraps) > data.parameters.iPositionResolution;
	iPositionMeasuredInconsistency.1 := ABS(data.Motor[2].rMetalStrapPos-data.Motor[2].rMeasuredDistanceMetalStraps) > data.parameters.iPositionResolution;

	IF iPositionMeasuredInconsistency>0 AND data.parameters.xPositionSensorInstalled AND xMotorStopped THEN
		data.Alarms.xPositionMeasuredInconsistency := TRUE;
	END_IF

	IF EDGEPOS(data.Alarms.xPositionMeasuredInconsistency) THEN
		rInputMeasuredDifference := (data.Motor[1].rMetalStrapPos-data.Motor[1].rMeasuredDistanceMetalStraps);
		rOutputMeasuredDifference := (data.Motor[2].rMetalStrapPos-data.Motor[2].rMeasuredDistanceMetalStraps);
	END_IF

	//Alarms summary
	//Stop
	iReasonStop.0 := data.Alarms.xMotorError;
	iReasonStop.1 := data.Alarms.xCommsMotorError;
	iReasonStop.2 := data.Alarms.xNotReferenced;
	iReasonStop.3 := xAnyMotorError;
	//iReasonStop.4 := data.Alarms.xPositionMeasuredInconsistency;

	data.AlSummary.xAlarmStop := iReasonStop > 0;
	IF EDGEPOS(data.AlSummary.xAlarmStop) THEN
		data.AlSummary.iReasonStop[0] := iReasonStop;
		LogStopAlarm;
	ELSIF EDGEPOS(NOT data.commands.AutoMode.xStop AND NOT data.AlSummary.xAlarmStop) THEN
		data.AlSummary.iReasonStop[0] := 0;
	END_IF

	//Critical
	iReasonCritical.0 := data.Alarms.xPositionOutOfRange;

	data.AlSummary.xAlarmCritical := iReasonCritical > 0;
	IF EDGEPOS(data.AlSummary.xAlarmCritical) THEN
		data.AlSummary.iReasonCritical := iReasonCritical;
		LogCriticalAlarm;
	ELSIF EDGEPOS(data.commands.Mode.xAuto AND NOT data.AlSummary.xAlarmCritical) THEN
		data.AlSummary.iReasonCritical := 0;
	END_IF

	//Warning
	// It is just used for drive alarms
	//iAnyWarning.0 := ;
	data.AlSummary.xAnyWarning:= iAnyWarning > 0;

	IF EDGEPOS(data.AlSummary.xAnyWarning) THEN
		data.AlSummary.iReasonWarning := iAnyWarning;
		LogWarningAlarm;
	ELSIF EDGEPOS(NOT data.AlSummary.xAnyWarning) THEN
		data.AlSummary.iReasonWarning := 0;
	END_IF

END_ACTION
```

#### AlarmSounds.st
```iecst
ACTION AlarmSounds:

	// Alarms reseteable sound management.
	ars_AlrStop.xAlarm:= data.AlSummary.xAlarmStop;
	ars_AlrStop.xSilence:= data.commands.xMute;
	ars_AlrStop();

	ars_AlrCritical.xAlarm:= data.AlSummary.xAlarmCritical;
	ars_AlrCritical.xSilence:= data.commands.xMute;
	ars_AlrCritical();

	ars_AlrWarning.xAlarm:= data.AlSummary.xAnyWarning;
	ars_AlrWarning.xSilence:= data.commands.xMute;
	ars_AlrWarning();

	data.AlSummary.xAlarmSound:= 	//ars_AlrWarning.xAlarmSound OR
									ars_AlrStop.xAlarmSound OR
									ars_AlrCritical.xAlarmSound OR
									(xAnyManualOrder AND gPLC.xBlk_200ms);

END_ACTION
```

#### ResetCommands.st
```iecst
ACTION ResetCommands:
	data.commands.xMoveBackward := FALSE;
	data.commands.xMoveForward  := FALSE;
	data.commands.xReference := FALSE;
END_ACTION
```

#### EventLog.st
```iecst
ACTION LogWarningAlarm:

	stWarningAlarmsLog.Source := ELOG_TYPE_PAIRED_ICLA;
	stWarningAlarmsLog.Severity:= ELOG_SEVERITY_INFO;
	stWarningAlarmsLog.Facility:= 0;
	stWarningAlarmsLog.ErrorCode:=0;

	stWarningAlarmsLog.Text := 'PairedIcla.LogWarningAlarm';

	IF iReasonWarning.0 THEN stWarningAlarmsLog.Text := 'data.Alarms.xReferencing';
	END_IF

	gEventLogLoader.EventData := ADR(stWarningAlarmsLog);
	gEventLogLoader();
END_ACTION

ACTION LogStopAlarm:

	stStopAlarmsLog.Source := ELOG_TYPE_PAIRED_ICLA;
	stStopAlarmsLog.Severity:= ELOG_SEVERITY_INFO;
	stStopAlarmsLog.Facility:= 0;
	stStopAlarmsLog.ErrorCode:=0;

	stStopAlarmsLog.Text := 'PairedIcla.LogStopAlarm';

	IF iReasonStop.0 THEN stStopAlarmsLog.Text := 'data.Alarms.xMotorError';
	ELSIF iReasonStop.1 THEN stStopAlarmsLog.Text := 'data.Alarms.xComsMotorError';
	ELSIF iReasonStop.2 THEN stStopAlarmsLog.Text := 'data.Alarms.xNotReferenced';
	END_IF

	gEventLogLoader.EventData := ADR(stStopAlarmsLog);
	gEventLogLoader();
END_ACTION

ACTION LogCriticalAlarm:

	stCriticalAlarmsLog.Source := ELOG_TYPE_PAIRED_ICLA;
	stCriticalAlarmsLog.Severity:= ELOG_SEVERITY_ERROR;
	stCriticalAlarmsLog.Facility:= 0;
	stCriticalAlarmsLog.ErrorCode:=0;

	stCriticalAlarmsLog.Text := 'PairedIcla.LogCriticalAlarm';

	IF iReasonCritical.0 THEN stCriticalAlarmsLog.Text := 'data.Alarms.xPositionOutOfRange';
//	ELSIF iReasonCritical.1 THEN stCriticalAlarmsLog.Text := '';
//	ELSIF iReasonCritical.2 THEN stCriticalAlarmsLog.Text := '';
//	ELSIF iReasonCritical.3 THEN stCriticalAlarmsLog.Text := '';
//	ELSIF iReasonCritical.4 THEN stCriticalAlarmsLog.Text := '';
//	ELSIF iReasonCritical.5 THEN stCriticalAlarmsLog.Text := '';
	END_IF

	gEventLogLoader.EventData := ADR(stCriticalAlarmsLog);
	gEventLogLoader();
END_ACTION
```

#### PairedIclaMotors.var - Local variables
```iecst
VAR
	data : REFERENCE TO PairedIclaMotors_typ;
	IclaMaster : REFERENCE TO stIcla;
	IclaGear : REFERENCE TO stIcla;
	IclaMotors : ARRAY[0..2] OF stIcla;
	stAlarmsReseted : PairedIclaMotorsAlarms;
	stAlarmSummaryReseted : stEFI_AlarmSummary;
END_VAR
VAR CONSTANT
	iHistoryLines : USINT := 20;
END_VAR
VAR
	IndexIclaMaster : USINT;
	IndexIclaGear : USINT;
	xAnyManualMovement : BOOL;
	rCopyPositionDesired : REAL;
	rPositionDesired : REAL;
	rPositionMotorMm : REAL;
	ars_AlrStop : AutoResetSound;
	ars_AlrCritical : AutoResetSound;
	ars_AlrWarning  : AutoResetSound;
	iReasonWarning : UDINT;
	iReasonStop : UDINT;
	iReasonCritical : UDINT;
	StateHistory : ARRAY[0..iHistoryLines] OF PairedIclaMotorsState;
	iIndexHistory : USINT;
	MotorDriveUnit : DriveUnitMngr;
	rJogSpeedSetPoint : REAL;
	xControllerReady : BOOL;
	xMotorsReferenced : BOOL;
	xMotorsInPosition : BOOL;
	xManualMovementEnabled : BOOL;
	xPoweredOn : BOOL;
	xMotorReady : BOOL;
	xAnyMotorError : BOOL;
	xAnyManualOrder : BOOL;
	iAnyAlarm : UINT;
	iAnyWarning : UINT;
	tonMotorStopped : TON;
	xReferencePositionReached : BOOL;
	xMotorStopped : BOOL;
	stCriticalAlarmsLog : EventLog_typ;
	stStopAlarmsLog : EventLog_typ;
	stWarningAlarmsLog : EventLog_typ;
	iIndexIclaMotor : USINT;
	iSystemState : PairedIclaMotorsState;
	iNumIclaMotors : USINT;
	iMisalignmentTolerance : USINT;
	rInterceptAnalogSensor : REAL := 58.0;
	rSlopeAnalogSensor : REAL := 0.0183;
	iPositionMeasuredInconsistency : USINT;
	rMeasuredDistanceMetalStraps : ARRAY[0..MAX_EHD_MOTORS_PER_ADJUST_SYS] OF REAL;
	rAnalogSensorTolerance : REAL := 0.4;
	rOutputMeasuredDifference : REAL;
	rInputMeasuredDifference : REAL;
END_VAR
```

### PairedIclaMotors.typ
```iecst
TYPE
	PairedIclaMotors_typ : 	STRUCT
		commands : PairedIclaMotorsCommands; (*Commands gui*)
		parameters : PairedIclaMotorsParameters; (*Parameters gui*)
		status : PairedIclaMotorsStatus; (*States potocell system*)
		Alarms : PairedIclaMotorsAlarms; (*Alarms*)
		AlSummary : stEFI_AlarmSummary; (*Alarms Summary*)
		Motor : ARRAY[0..2]OF PairedIclaMotors_Motor;
		Inputs : PairedIclaInputs;
	END_STRUCT;
	PairedIclaMotors_Motor : 	STRUCT
		Inputs : PairedIclaMotorsInputs;
		Icla : stIcla;
		Alarms : MotorAlarms;
		iDirection : INT; (*1= Clockwise, -1=Conterclockwise*)
		rHomePosition : REAL;
		rMotorResolution : REAL;
		rDistanceFromSensorTargetToStrap : REAL := 10; (*Distance From Sensor Target To metal Strap*)
		rDistanceBetweenSensors : REAL;
		rMeasuredDistanceMetalStraps : REAL;
		rMeasuredPositionFrontSide : REAL; (*Position in mm of the motors on front/user side*)
		rMeasuredPositionBackSide : REAL; (*Position in mm of the motors on back/electrical cabinet side*)
		rPositionMotor : REAL; (*Position in mm of the motors*)
		rMetalStrapPos : REAL; (*Position in mm of the metal straps using motor information*)
	END_STRUCT;
	PairedIclaMotorsCommands : 	STRUCT
		xMoveForward : BOOL;
		xMoveBackward : BOOL;
		xReference : BOOL;
		xErrorRst : BOOL;
		xMute : BOOL;
		AutoMode : stEFI_MachineAutoModes;
		Mode : StGeneral_States_Mode;
		xStop : BOOL;
		xResetMotor : BOOL;
	END_STRUCT;
	PairedIclaMotorsParameters : 	STRUCT
		xEnabled : BOOL;
		xMovementsEnabled : BOOL;
		xInstalled : BOOL; (*This variable is activated when this functionality is intalled and ready to be enabled*)
		xPositionSensorInstalled : BOOL; (*This variable is activated when motors positions are measured in addition to internal encoder position calculation*)
		DriveUnit : MC_DriveUnitManager;
		IndexIclaMaster : USINT; (*Index of the motor in gAxis array*)
		IndexIclaGear : USINT; (*Index of the motor in gAxis array*)
		rPositionDesired : REAL;
		rMechPositionMin : REAL; (*Mechanical max position allowed*)
		rMechPositionMax : REAL; (*Mechanical max position allowed*)
		Acceleration : REAL := 5; (*Acc SP mm/ s2*)
		JogSpeed : REAL := 10; (*Jog Speed SP mm/s*)
		Speed : REAL := 100; (*Speed SP mm/s*)
		iNumIclaMotors : USINT := 2; (*Number of motors used in this adjustment system*)
		rDistanceFromSensorToBeltsCenter : REAL := 116; (*rDistance From Sensor To Belts Center. Same value for both entry and exit side*)
		rMaxPositionMeasured : REAL := 600; (*Max position measured by sensor*)
		iPositionResolution : REAL := 2; (*Position resolution in mm*)
		iMisalignmentTolerance : USINT;
	END_STRUCT;
	PairedIclaMotorsStatus : 	STRUCT
		xEnabled : BOOL;
		xInstalled : BOOL;
		xReferencing : BOOL;
		xReferenced : BOOL;
		xMoving : BOOL; (*Motors are moving*)
		xInPosition : BOOL; (*Motors are positioned on desired position*)
		iSystemState : PairedIclaMotorsState := NOT_INITIALIZED;
	END_STRUCT;
	PairedIclaMotorsAlarms : 	STRUCT
		xNotReferenced : BOOL; (*Phocell system not homed*)
		xNotInstalled : BOOL;
		xCommsMotorError : BOOL;
		xMotorError : BOOL; (*Error Id != 0*)
		xNotAligned : BOOL; (*Motors are not at the same position*)
		xPositionMeasuredInconsistency : BOOL; (*Inconsistency between position measured (analogic input) and motor position information (motors encoder)*)
		xPositionOutOfRange : BOOL; (*Motor is positioned out of mechanical range allowed*)
		xControllerNotReady : BOOL; (*Waiting for enable input (STO_A, STO_B)*)
	END_STRUCT;
	PairedIclaMotorsState :
		(
		NOT_USED,
		NOT_INITIALIZED,
		POWER_ON,
		HOME_DIR,
		POWERED,
		HOMING_STEP_1,
		HOMING_STEP_2,
		HOMING_STEP_3,
		STANDSTILL,
		MANUAL,
		JOGGING,
		AUTO,
		RUNNING,
		ERROR
		);
	PairedIclaMotorsInputs : 	STRUCT
		xMaxPositionReached : BOOL; (*Maximum position feedback received from an inductive sensor*)
		xMinPositionReached : BOOL; (*Minimum position feedback received from an inductive sensor*)
		xMeasuredPositionFrontSideError : BOOL; (*analogic sensor error*)
		iMeasuredPositionFrontSide : INT; (*Position feedback receive from an analogic sensor*)
		xMeasuredPositionBackSideError : BOOL; (*analogic sensor error*)
		iMeasuredPositionBackSide : INT; (*Position feedback receive from an analogic sensor*)
	END_STRUCT;
	MotorAlarms : 	STRUCT
		xCommsMotorError : BOOL;
		xMotorError : BOOL; (*Error Id != 0*)
		xControllerNotReady : BOOL; (*Waiting for enable input (STO_A, STO_B)*)
	END_STRUCT;
	PairedIclaInputs : 	STRUCT
		xSafetyEnable : BOOL;
	END_STRUCT;
END_TYPE
```

### InitPairedIclaMotorsSim.var
```iecst
VAR
	iPairedIclaMotorSimIndex : USINT;
END_VAR
```

- Program Logical/ExtPack/_Transport/PairedIclaMotors/PairedIclaMotorsSim/PairedIclaMotorsSim_v1/InitPairedIclaMotorsSim (IEC) (no source held here)

### Program Logical/ExtPack/_Transport/PairedIclaMotors/PairedIclaMotorsSim/PairedIclaMotorsSim_v1/PairedIclaMotorsSim

#### PairedIclaMotorsSim.var
```iecst
VAR
	data : REFERENCE TO PairedIclaMotors_typ;
	tonHoming : TON;
END_VAR
```

#### PairedIclaMotorsSim.st
```iecst
PROGRAM _INIT
	(* Insert code here *)

END_PROGRAM

PROGRAM _CYCLIC
	(* Insert code here *)
	data ACCESS ADR (gPairedMotors[iPairedIclaMotorSimIndex]);

	tonHoming.IN := data.status.iSystemState = HOMING_STEP_1;
	tonHoming.PT := t#1s;
	tonHoming();
	IF tonHoming.Q THEN
		data.Motor[1].Inputs.xMinPositionReached := TRUE;
		data.Motor[2].Inputs.xMinPositionReached := TRUE;

	ELSIF data.status.xReferenced THEN
		//Min position sensors
		data.Motor[1].Inputs.xMinPositionReached := (data.Motor[1].rPositionMotor<data.parameters.rMechPositionMin);
		data.Motor[2].Inputs.xMinPositionReached := (data.Motor[2].rPositionMotor<data.parameters.rMechPositionMin);

		//Max position sensors
		data.Motor[1].Inputs.xMaxPositionReached := (data.Motor[1].rPositionMotor>data.parameters.rMechPositionMax);
		data.Motor[2].Inputs.xMaxPositionReached := (data.Motor[2].rPositionMotor>data.parameters.rMechPositionMax);

		IF data.parameters.xPositionSensorInstalled THEN
			data.Motor[1].Inputs.iMeasuredPositionFrontSide := data.Motor[1].Inputs.iMeasuredPositionBackSide := REAL_TO_INT((data.Motor[1].rPositionMotor * 16384 / 600) + 16383);
			data.Motor[2].Inputs.iMeasuredPositionFrontSide := data.Motor[2].Inputs.iMeasuredPositionBackSide := REAL_TO_INT((data.Motor[2].rPositionMotor * 16384 / 600) + 16383);
		END_IF

	END_IF

	iPairedIclaMotorSimIndex := iPairedIclaMotorSimIndex + 1;

END_PROGRAM

PROGRAM _EXIT
	(* Insert code here *)

END_PROGRAM
```

### Program Logical/ExtPack/_Transport/BeltCleaning/BeltCleaning_v1/BeltCleaning (IEC)

#### BeltClean.var
```iecst
VAR
	ResetOutputs : BeltCleanOutputs_typ;
	ResetCommands : BeltCleanCommands_typ;
	ResetCommandsSw : BeltCleanCommandsSw_typ;
	dataBeltClean : REFERENCE TO BeltClean_typ;
	iReasonStop : UINT;
	tofCleaningSystemRise : TOF;
	tonCleanBeltPump : TON;
	tonCleaningByTime : TON;
	xEdge1sec : BOOL;
	ResetAlarms : BeltCleanAlarm_typ;
	ResetAlSummary : stEFI_AlarmSummary;
	ton_Cleaning : TON;
	ton_Drying : TON;
	ars_AnyAlarm : AutoResetSound;
	ton_SwCleanRequest : TON;
	ton_CleanRequest : TON;
	iTimeElapsed : UDINT;
	iPieces : UDINT;
	ton_WaitingToCleanState : TON;
END_VAR
```

#### Alarms.st
```iecst
ACTION Alarms:

	//WARNING
	IF NOT dataBeltClean.ParSw.xAirTurbineEnabled THEN
		dataBeltClean.Alarm.xAirTurbDisabled := TRUE;
	END_IF
	IF NOT dataBeltClean.Inputs.xAirTurbVSDAvailable THEN
		dataBeltClean.Alarm.xAirTurbDisVSDFault := TRUE;
	END_IF
	IF dataBeltClean.Commands.xAcceptRequest AND NOT dataBeltClean.Parameters.xBeltEmpty THEN
		dataBeltClean.Alarm.xBeltNotEmptyToClean := TRUE;
	END_IF

	//STOP
	IF (dataBeltClean.Status.State = BCLEAN_CLEANING OR dataBeltClean.Status.State = BCLEAN_DRYING) AND NOT dataBeltClean.Parameters.xBeltRunning THEN
		dataBeltClean.Alarm.xBeltIsNotRuning := TRUE;
	END_IF
	IF dataBeltClean.ParSw.xAirTurbineEnabled AND NOT dataBeltClean.Inputs.xAirTurbVSDAvailable THEN
		dataBeltClean.Alarm.xAirTurbEnVSDFault := TRUE;
	END_IF
	IF ton_WaitingToCleanState.Q THEN
		dataBeltClean.Alarm.xWaitingToCleanState := TRUE;
	END_IF

	IF dataBeltClean.Status.xCleaning AND NOT dataBeltClean.Parameters.xBeltEmpty THEN
		dataBeltClean.Alarm.xBeltIsNotEmpty := TRUE;
	END_IF

END_ACTION
```

#### GeneralLogic.st
```iecst
ACTION GeneralLogic:

	//Cleaning Belt by time. When cleaning, the time is reseted
	IF dataBeltClean.ParSw.xEnabledByTime AND dataBeltClean.Status.State = BCLEAN_ENABLED AND dataBeltClean.Parameters.Mode.xAuto THEN
		xEdge1sec := EDGEPOS(gPLC.xBlk_1s);
		IF dataBeltClean.Parameters.xBeltRunning AND xEdge1sec THEN
			iTimeElapsed := iTimeElapsed + 1;
		END_IF
		IF iTimeElapsed > dataBeltClean.ParSw.iTimeToClean  THEN
			dataBeltClean.Status.xCleanReqByTime := TRUE;
		END_IF
		dataBeltClean.Status.iTimeToClean := dataBeltClean.ParSw.iTimeToClean - iTimeElapsed;
	END_IF

	// Tiles counter
	IF dataBeltClean.ParSw.xEnabledByPieces AND dataBeltClean.Status.State = BCLEAN_ENABLED AND dataBeltClean.Parameters.Mode.xAuto THEN
		IF EDGEPOS (dataBeltClean.Inputs.xEnteringMedia) THEN
			iPieces := iPieces + 1;
		END_IF

		IF iPieces >= dataBeltClean.ParSw.iPiecesToClean THEN
			dataBeltClean.Status.xCleanReqByPieces := TRUE;
		END_IF
		dataBeltClean.Status.iPiecesToClean := dataBeltClean.ParSw.iPiecesToClean - iPieces;
	END_IF

	// Request activation
	dataBeltClean.Status.xCleanForced := dataBeltClean.CommandsSw.xClean;

	//ResetCountersAndTimers
	IF dataBeltClean.CommandsSw.xResetCounters AND dataBeltClean.Status.State = BCLEAN_DISABLED THEN
		ResetCountersAndTimers;
	END_IF

	//Sw request timer
	ton_SwCleanRequest.IN := dataBeltClean.Status.State = BCLEAN_WAITING_SW_CONF;
	ton_SwCleanRequest.PT := T#120s;
	ton_SwCleanRequest();

	//Waiting request to clean accepted
	ton_WaitingToCleanState.IN := dataBeltClean.Status.State = BCLEAN_WAITING_TO_CLEAN;
	ton_WaitingToCleanState.PT := T#5m;
	ton_WaitingToCleanState();

	//State timers
	ton_Cleaning.IN := dataBeltClean.Status.State = BCLEAN_CLEANING;
	ton_Cleaning.PT :=dataBeltClean.ParSw.tiCleaning;
	ton_Cleaning();

	ton_Drying.IN := dataBeltClean.Status.State = BCLEAN_DRYING;
	ton_Drying.PT := dataBeltClean.ParSw.tiDrying;
	ton_Drying();

	//Delay falling the tray to be sure no water is poured inside the machine
	tofCleaningSystemRise.IN:= dataBeltClean.Status.State = BCLEAN_CLEANING;
	tofCleaningSystemRise.PT:=T#200MS;
	tofCleaningSystemRise();

	//Delay pneumatic pump to avoid pouring water inside the machine
	tonCleanBeltPump.IN:= dataBeltClean.Status.State = BCLEAN_CLEANING;
	tonCleanBeltPump.PT:=T#900ms;
	tonCleanBeltPump();

END_ACTION

ACTION ResetCountersAndTimers:

	dataBeltClean.Status.iTimeToClean := 0;
	iTimeElapsed := 0;
	dataBeltClean.Status.iPiecesToClean := 0;
	iPieces := 0;
	dataBeltClean.Status.xCleanReqByPieces := FALSE;
	dataBeltClean.Status.xCleanReqByTime := FALSE;
	dataBeltClean.Status.xCleanForced := FALSE;

END_ACTION
```

#### Outputs.st
```iecst
ACTION Outputs:

	IF dataBeltClean.Parameters.Mode.xZero THEN
		dataBeltClean.Outputs := ResetOutputs;

	ELSIF dataBeltClean.Parameters.Mode.xManual THEN
		dataBeltClean.Outputs.xRiseCleaningSystem := dataBeltClean.Orders.Manual.xToCleanPosition;
		dataBeltClean.Outputs.xPumpOn := dataBeltClean.Orders.Manual.xRunPump;
		dataBeltClean.Outputs.xAirTurbineOn := dataBeltClean.Orders.Manual.xRunAirTurbine AND dataBeltClean.ParSw.xAirTurbineEnabled;

	ELSIF dataBeltClean.Parameters.Mode.xAuto THEN
		dataBeltClean.Outputs.xRiseCleaningSystem := dataBeltClean.Status.State = BCLEAN_CLEANING AND tofCleaningSystemRise.Q;
		dataBeltClean.Outputs.xPumpOn := dataBeltClean.Status.State = BCLEAN_CLEANING AND tonCleanBeltPump.Q;
		dataBeltClean.Outputs.xAirTurbineOn := (dataBeltClean.Status.State = BCLEAN_CLEANING OR dataBeltClean.Status.State = BCLEAN_DRYING) AND dataBeltClean.ParSw.xAirTurbineEnabled;

	END_IF

	dataBeltClean.Outputs.xAirTurbineVSDReset := dataBeltClean.ParSw.xAirTurbineEnabled AND dataBeltClean.Commands.xReset;

END_ACTION
```

### BeltClean.typ - Local data types
```iecst
TYPE
	BeltCleanState_enum :
		(
		BCLEAN_NOT_INSTALLED, (*Belt clean system not installed*)
		BCLEAN_FAULT, (*Belt clean system in fault*)
		BCLEAN_DISABLED, (*Belt clean system disabled*)
		BCLEAN_ENABLED, (*Belt clean system enabled*)
		BCLEAN_WAITING_SW_CONF, (*Waiting SW confirmation to clean*)
		BCLEAN_WAITING_TO_CLEAN, (*Beltl Clean system waiting accept request to clean*)
		BCLEAN_CLEANING, (*Belt Clean system cleaning with water and air if enabled*)
		BCLEAN_DRYING (*Belt Clean system drying only*)
		);
	BeltCleanParam_typ : 	STRUCT
		Mode : StGeneral_States_Mode;
		xBeltRunning : BOOL; (*Belt is runing*)
		rBeltSpeed : REAL; (*Belt speed*)
		xBeltEmpty : BOOL; (*Belt is empty*)
		xInstalled : BOOL; (*Water belt clean system installed*)
	END_STRUCT;
	BeltCleanCommandsSw_typ : 	STRUCT
		xResetCounters : BOOL; (*Command to reset counters*)
		xClean : BOOL; (*To directly request a clean from UI*)
		xRefuseRequest : BOOL; (*UI command to refuse the request to clean*)
		xAcceptRequest : BOOL; (*UI command to accept the request to clean*)
	END_STRUCT;
	BeltCleanCommands_typ : 	STRUCT
		xReset : BOOL; (*Alarm reset*)
		xMute : BOOL; (*Mute alarm*)
		xAcceptRequest : BOOL; (*Accepted request to clean*)
	END_STRUCT;
	BeltCleanOrders_typ : 	STRUCT
		Manual : BeltCleanOrdersManual_typ; (*Manual movements*)
	END_STRUCT;
	BeltCleanOrdersManual_typ : 	STRUCT
		xRunPump : BOOL; (*Run pump in manual mode*)
		xRunAirTurbine : BOOL; (*Run air turbine in manual mode*)
		xToCleanPosition : BOOL; (*Move cleaning system to cleaning position*)
	END_STRUCT;
	BeltCleanOutputs_typ : 	STRUCT
		xAirTurbineVSDReset : BOOL; (*Air turbine VSD reset*)
		xAirTurbineOn : BOOL; (*Start air turbine*)
		xPumpOn : BOOL; (*Start pump*)
		xRiseCleaningSystem : BOOL; (*Rise cleaning system to cleaning position*)
	END_STRUCT;
	BeltCleanStatus_typ : 	STRUCT
		State : BeltCleanState_enum;
		xEnabled : BOOL;
		xCleaning : BOOL; (*Cleaning or drying is being performed*)
		iPiecesToClean : UDINT; (*Number of pieces left to next clean*)
		iTimeToClean : UDINT; (*Time left to next clean*)
		xCleanReqByTime : BOOL; (*Cleaning required by time*)
		xCleanReqByPieces : BOOL; (*Cleaning required by pieces*)
		xCleanForced : BOOL; (*Cleaning required by UI*)
		xCleanRequestedSw : BOOL; (*Cleaning request to UI*)
		xCleanRequested : BOOL; (*Clean requested to machine*)
	END_STRUCT;
	BeltCleanAlarm_typ : 	STRUCT
		xAirTurbDisabled : BOOL; (*Air turbine disabled from UI*)
		xAirTurbDisVSDFault : BOOL; (*Air turbine disabled from UI and VSD in fault*)
		xAirTurbEnVSDFault : BOOL; (*Air turbine enabled from UI and VSD in fault*)
		xBeltIsNotRuning : BOOL; (*Belt not running while cleaning or drying*)
		xWaitingToCleanState : BOOL; (*Waiting to accept request for more than 5 minutes*)
		xBeltIsNotEmpty : BOOL; (*Belt is not empty while belt cleaning*)
		xBeltNotEmptyToClean : BOOL; (*Belt not empty when start belt cleaning was requested*)
	END_STRUCT;
	BeltCleanInputs_typ : 	STRUCT
		xEnteringMedia : BOOL; (*Media entering into machine*)
		xAirTurbVSDAvailable : BOOL; (*Air turbine VSD available*)
	END_STRUCT;
	BeltCleanParSw_typ : 	STRUCT
		xAirTurbineEnabled : BOOL; (*Air turbine drying enabled*)
		xEnabledByTime : BOOL; (*Cleaning by time enabled*)
		xEnabledByPieces : BOOL; (*Cleaning by pieces enabled*)
		rCleanBeltSpeed : REAL := 20.0; (*Belt speed while cleaning*)
		iTimeToClean : UDINT; (*Number of seconds between cleanings*)
		iPiecesToClean : UDINT; (*Number of pieces between cleanings*)
		tiCleaning : TIME := T#120s; (*Duration of cleaning step*)
		tiDrying : TIME := T#60s; (*Duration of drying step*)
	END_STRUCT;
	BeltClean_typ : 	STRUCT
		Commands : BeltCleanCommands_typ;
		CommandsSw : BeltCleanCommandsSw_typ;
		Orders : BeltCleanOrders_typ;
		Inputs : BeltCleanInputs_typ;
		Parameters : BeltCleanParam_typ;
		ParSw : BeltCleanParSw_typ;
		Status : BeltCleanStatus_typ;
		AlSummary : stEFI_AlarmSummary;
		Alarm : BeltCleanAlarm_typ;
		Outputs : BeltCleanOutputs_typ;
	END_STRUCT;
END_TYPE
```

### Program Logical/ExtPack/_Transport/BeltCleaning/BeltCleaningSim/BeltCleaningSim (IEC)

#### BeltCleanSim.var
```iecst
VAR
	BeltClean : REFERENCE TO BeltClean_typ;
END_VAR
```

### Package Logical/ExtPack/_Extras/ChillerCtrl/ChillerCtrl_v2 - Icla Ctrl Logic package

### Program Logical/ExtPack/_Extras/ChillerCtrl/ChillerCtrl_v2/InitChiller (IEC)

#### InitChiller.st
```iecst
PROGRAM _CYCLIC
	iIndexChiller:=1;
END_PROGRAM
```

### Program Logical/ExtPack/_Extras/ChillerCtrl/ChillerCtrl_v2/ChillerCtrl (IEC)

#### Chiller.st
```iecst
PROGRAM _CYCLIC

	// Assigning dataChillConfig to determine the Configuration of the Chilled and the Chiller Type
	dataChill ACCESS ADR (gChiller[iIndexChiller]);

	// Currently we do not have any confirmation the chiller is installed
	dataChill.St.xInstalled := dataChill.Parameters.xInstalled;

	dataChill.St.xEnabled := dataChill.parSw.xEnable OR dataChill.Parameters.xEnable;

	IF NOT dataChill.St.xInstalled OR NOT dataChill.St.xEnabled THEN
		ResetAlarms;
		iIndexChiller:= iIndexChiller +1;
		RETURN;
	END_IF

	Conversions;
	StateCtrl;
	alarms;
	alarmsSound;
	alarmsSummary;

	iIndexChiller := iIndexChiller + 1;

END_PROGRAM
```

#### ChillerCtrl.st
```iecst
ACTION StateCtrl:

	CASE ChillerState OF

		CHILLER_OFF:
			IF xRunOrder THEN
				ChillerState := CHILLER_STARTING;
			END_IF

		CHILLER_STARTING:
			IF dataChill.In.xPowered THEN
				ChillerState := CHILLER_RUNNING;
			END_IF

			IF NOT xRunOrder THEN
				ChillerState := CHILLER_STOPPING;
			END_IF

		CHILLER_RUNNING:
			IF NOT xRunOrder THEN
				ChillerState := CHILLER_STOPPING;
			END_IF

		CHILLER_STOPPING:
			IF TON_DelayChillerStopped.Q THEN
				ChillerState := CHILLER_OFF;
			END_IF

		CHILLER_FAULT:
			ResetRunCommands;
			IF NOT dataChill.In.xAlarm THEN
				ChillerState := CHILLER_STARTING;
			END_IF

	END_CASE

	//Timer chiller stopping
	CASE dataChill.Parameters.SystemType OF
		CHILLERSYS_DIRECT:
			TON_DelayChillerStopped.PT:= T#1h;
		CHILLERSYS_WATERMANIFOLD:
			TON_DelayChillerStopped.PT:= T#30s;
		ELSE
			TON_DelayChillerStopped.PT:= T#300s;
	END_CASE

	TON_DelayChillerStopped.IN := (ChillerState = CHILLER_STOPPING);
	TON_DelayChillerStopped();

	iReasonRunning.0 := ChillerState = CHILLER_RUNNING;
	iReasonRunning.1 := ChillerState = CHILLER_STARTING;
	iReasonRunning.2 := ChillerState = CHILLER_STOPPING;
	tonChillerRunning.IN := iReasonRunning > 0 ;
	tonChillerRunning.PT := T#15s;
	tonChillerRunning();

	IF tonChillerRunning.Q AND dataChill.Alarm.xInAlarm THEN
		ChillerState := CHILLER_FAULT;
	END_IF

	// Define the particular RUN signal
	CASE dataChill.Parameters.SystemType OF
		CHILLERSYS_DIRECT:
			xRunOrder := dataChill.Orders.xRun;
		CHILLERSYS_WATERMANIFOLD:
			WaterManifoldCtrl;
			xRunOrder := dataChill.Orders.xRun OR xManifoldRunOrder;
	END_CASE

	dataChill.St.xRunning := iReasonRunning > 0;
	dataChill.Out.xStart := dataChill.St.xRunning;
	dataChill.St.Status := ChillerState;

END_ACTION

ACTION WaterManifoldCtrl:

	//ON conditions//
	xNeedCold := dataChill.St.WaterManifold.rManifoldTemp > (dataChill.Parameters.rTempSetPoint-LC_OFFSET_TEMP_TO_START_STOP);

	tonChillerON.IN:= xNeedCold AND dataChill.Orders.xRun;
	tonChillerON.PT:= t#20s;
	tonChillerON();

	//OFF conditions//
	xEnoughCold := dataChill.St.WaterManifold.rManifoldTemp < (dataChill.Parameters.rTempSetPoint-LC_OFFSET_TEMP_TO_START_STOP);

	tonChillerOFF.IN:= xEnoughCold OR NOT dataChill.Orders.xRun;
	tonChillerOFF.PT:=t#20s;
	tonChillerOFF();

	//Revisar si esto ha funcionado alguna vez, porque la antigua orden de xAnyRunOrder estaba supeditada a la orden de run que viene de machinectrlslow (basicamente cuando cualquier sistema de tintas esta en marcha
	//y en paralelo, a esta de Run que se activa a continuación si es watermanifold, pero es que el rTempSetPoint salta a 100ºC si no hay ninguna barra encendida, así que esto de watermanifold no sirve de nada.
	IF tonChillerON.Q THEN
		xManifoldRunOrder := TRUE;
	ELSIF tonChillerOFF.Q THEN
		xManifoldRunOrder := FALSE;
	END_IF

END_ACTION

ACTION ResetRunCommands:

	xManifoldRunOrder := FALSE;

END_ACTION
```

### Chiller Doc.txt - Documentation for using the package
```
#################################################################################
#################################################################################
#
#						GENERAL USE OF CHILLERCTRL PACKAGE
#
# 	To use this package unit, some general input variables are needed:
#	dataChill as 	gChillerInks[iIndexChiller]
#	-dataChill.In.xStopChiller: It is the signal to stop chiller, its activated when the system
#	to control temperature doen't need it (Inks stopped or PH without power).
#	-dataChill.In.xChillerWorking: Chiller working feedback from physicall machine.
# 	-dataChill.In.iTempEnvironment: is the environment temp.measured with a gauge.
#	-dataChill.In.iWaterCollectorTemp: temperature at the exit collector of the chiller.
# 	-dataChill.In.xTempEnvSensError: Emperature sensor error.
# 	-dataChill.In.xTempWatSensError: Emperature sensor error.
# 	-dataChill.In.xNoPowered: Signal from Chiller CB for report to SW CB problem, its warning alarm.
# 	-dataChill.In.rControledTemp: Temperature to control.
#################################################################################
						ON/OFF CONDITIONS AND CONTROL
	The outputs of the package is:
	-dataChill.Out.xStart: Its true when:
	"dataChill.In.iTempEnvironment>(dataChill.Pt.rTempSetPoint-LC_OFFSET_TEMP_TO_START_STOP)" for 20 seconds OR
	when we force "dataChill.commands.xCoolingNeeded" (ready but not activate by program or by SW for the moment)
	and dont have any alarm in chiller, and its chage to false when:
	"dataChill.In.iTempEnvironment<(dataChill.Pt.rTempSetPoint-LC_OFFSET_TEMP_TO_START_STOP)" or Stop chiller order are active
	 if it's TRUE, the ON signal to chiller is sent.

#################################################################################
#################################################################################
#									ALARMS:
#	-dataChill.Al.Warning.xChillerNotWorking: set id chiller ON signal and the "dataChill.In.xChillerWorking" its nbot active.
#	-dataChill.Warning.xCheckChiller: Is used to send a message in UI to inform that the set point
#	must be changed manually in chiller. It is true when:
#	"(dataChill.Pt.rTempSetPoint < dataChill.In.rControledTemp)AND dataChill.Pt.xControlledSysNotHeating AND NOT dataChill.St.xChillerInAlarm"
#	-dataChill.Warning.xChillerInAlarm: its active when the alarm input are active
#	-dataChill.Warning.xAlrEnvTempSensBrokn & dataChill.Warning.xAlrTempSensBrokn:its active when the temperature sensor error input are active
#################################################################################
```

### Chiller.var
```iecst
VAR
	iIndexChiller : USINT;
END_VAR
```

### Program Logical/ExtPack/_Extras/ChillerCtrl/ChillerSim/ChillerSim_v1/ChillerSim (IEC)

#### Main.st - Init, cyclic, exit code
```iecst
PROGRAM _INIT
	(* Insert code here *)
	FOR iChillerSimIndex:=1 TO MAX_LAST_CHILLER DO
		// Referencing chiller
		dataChill ACCESS ADR(gChiller[iChillerSimIndex]);

		// Initial values
		dataChill.In.xAlarm := FALSE;
		dataChill.In.WaterManifold.xTempEnvSensError := FALSE;
		dataChill.In.WaterManifold.xTempWatSensError := FALSE;
	END_FOR

	simTemp.rA:= -0.0002;
	simTemp.rB:= -0.01;
	simTemp.rInitialValue:= 210;
	simTemp.rMinValue:= 160;
	simTemp.rMaxValue:= 320;

END_PROGRAM

PROGRAM _CYCLIC
	(* Insert code here *)
	dataChill ACCESS ADR(gChiller[iChillerSimIndex]);
	SimChiller ACCESS ADR(gSimChiller[iChillerSimIndex]);

	IF EDGEPOS(SimChiller.Commands.StopRunning) THEN
		SimChiller.Commands.StopRunning := FALSE;
		xChillerStopped := TRUE;
		dataChill.In.xPowered := FALSE;
	ELSE
		IF EDGEPOS(dataChill.Out.xStart) THEN
			xChillerStopped := FALSE;
		END_IF
		tonSignalRun.IN := dataChill.Out.xStart AND NOT xChillerStopped;
		tonSignalRun.PT := T#3s;
		tonSignalRun();
		dataChill.In.xPowered := tonSignalRun.Q;
		dataChill.In.xCooling := tonSignalRun.Q;

	END_IF

	dataChill.In.xAlarm := SimChiller.Commands.GenerateAlarm;

	IF dataChill.Out.xStart AND NOT dataChill.In.xAlarm THEN
		simTemp.rActionControl := 0.05;
	ELSE
		simTemp.rActionControl := 0;
	END_IF
	simTemp();
	dataChill.In.WaterManifold.iWaterManifoldTempRaw := REAL_TO_INT(simTemp.rPresentValue);

	dataChill.In.WaterManifold.iEnvironmentTempRaw := REAL_TO_INT(280);

	iChillerSimIndex := iChillerSimIndex + 1;

END_PROGRAM
```

#### ChillerSim.var - Local variables
```iecst
VAR
	SimChiller : REFERENCE TO stChillerSim;
	dataChill : REFERENCE TO StChiller;
	tonSignalRun : TON;
	xChillerStopped : BOOL;
	simTemp : SimAnalogProcess; (*Function block to simulate the temperature of the inks*)
END_VAR
```

### Program Logical/ExtPack/_Extras/ChillerCtrl/ChillerSim/ChillerSim_v1/InitChillerSim

#### Main.st
```iecst
PROGRAM _CYCLIC
	(* Init Index for Simulation *)
	iChillerSimIndex:=1;
END_PROGRAM
```

### PowerMeterCtrl.typ
```iecst
TYPE
	PowerMeterInputs_typ : 	STRUCT
		Comms : PowerMeterCommsInputs_typ;
	END_STRUCT;
	stPowerMeter : 	STRUCT
		Inputs : PowerMeterInputs_typ;
		Alarms : PowerMeterAlarms_typ;
		Status : PowerMeterStatus_typ;
		Parameters : PowerMeterParameters_typ;
		Commands : PowerMeterCommands_typ;
	END_STRUCT;
	PowerMeterCommsInputs_typ : 	STRUCT
		EffectiveCurrentPhaseA : UINT;
		EffectiveCurrentPhaseB : UINT;
		EffectiveCurrentPhaseC : UINT;
		EffectiveCurrentNeutral : UINT;
		MaxCurrentAllPhases : UINT;
		IgEarthDefectiveCurrent : UINT;
		CurrentDifferential : UINT;
		MaxEffectiveCurrentPhaseA : UINT;
		MaxEffectiveCurrentPhaseB : UINT;
		MaxEffectiveCurrentPhaseC : UINT;
		MaxEffectiveCurrentNeutral : UINT;
		MaxIgEarthDefectiveCurrent : UINT;
		MaxCurrentDifferential : UINT;
		EffectiveVoltagePhasesAB : UINT;
		EffectiveVoltagePhasesBC : UINT;
		EffectiveVoltagePhasesCA : UINT;
		EffectiveVoltagePhasesAN : UINT;
		EffectiveVoltagePhasesBN : UINT;
		EffectiveVoltagePhasesCN : UINT;
		Frequency : UINT;
		FrequencyMax : UINT;
		ActivePowerPhaseA : INT;
		ActivePowerPhaseB : INT;
		ActivePowerPhaseC : INT;
		TotalActivePower : INT;
		ApparentPowerPhaseA : INT;
		ApparentPowerPhaseB : INT;
		ApparentPowerPhaseC : INT;
		TotalApparentPower : UINT;
		ReactivePowerPhaseA : UINT;
		ReactivePowerPhaseB : UINT;
		ReactivePowerPhaseC : UINT;
		TotalReactivePower : UINT;
		THDVoltageAB : UINT;
		THDVoltageBC : UINT;
		THDVoltageCA : UINT;
		THDVoltageAN : UINT;
		THDVoltageBN : UINT;
		THDVoltageCN : UINT;
		THDCurrentA : UINT;
		THDCurrentB : UINT;
		THDCurrentC : UINT;
		TotalTHDCurrent : UINT;
		ReceivedDataModPowerMeter : ARRAY[0..120]OF UINT;
	END_STRUCT;
	PowerMeterAlarms_typ : 	STRUCT
		xCriticalAlarm : BOOL;
		xWarningAlarm : BOOL;
		xAnyAlarm : BOOL;
		xCommsError : BOOL;
	END_STRUCT;
	PowerMeterCommsStatus_typ : 	STRUCT
		xModuleOk : BOOL;
		ModSlaveState : UINT;
		LastError : UINT;
		LastErrorBlockNum : UINT;
		xStopButtonPressed : BOOL;
		ActOverloadError : BOOL;
		ActModbusError : BOOL;
		ActSlvConError : BOOL;
		ActRefreshError : BOOL;
		ActInternalError : BOOL;
		ActConfError : BOOL;
		HistOverloadError : BOOL;
		HistModbusError : BOOL;
		HistSlvConError : BOOL;
		HistRefreshError : BOOL;
		HistInternalError : BOOL;
		HistConfError : BOOL;
		ModbusErrorCnt : UINT;
		ModbusConErrorCnt : UINT;
		ModbusPktRefreshTimeoutCnt : UINT;
		ModbusPktPendPerSec : UINT;
		ModbusMeanResponseTime : UINT;
	END_STRUCT;
	PowerMeterStatus_typ : 	STRUCT
		Comms : PowerMeterCommsStatus_typ;
	END_STRUCT;
	PowerMeterParameters_typ : 	STRUCT
		xInstalled : BOOL; (*The powermeter is installed in the machine*)
		xActiveSlaveDiagnosis : BOOL;
	END_STRUCT;
	PowerMeterCommands_typ : 	STRUCT
		xMute : BOOL;
		xReset : BOOL;
	END_STRUCT;
END_TYPE
```

### PowerMeter.var
```iecst
VAR
	iIndexPowerMeter : USINT;
END_VAR
```

### Program Logical/ExtPack/_Extras/PowerMeterCtrl/PowerMeterCtrl_v1/InitPowerMeterCtrl

#### InitPowerMeterCtrl.st
```iecst
PROGRAM _CYCLIC
	iIndexPowerMeter := 1;
END_PROGRAM
```

### Program Logical/ExtPack/_Extras/PowerMeterCtrl/PowerMeterCtrl_v1/PowerMeterCtrl (IEC)

#### PowerMeter.st - Init, cyclic, exit code
```iecst
PROGRAM _CYCLIC

	PowerMeter ACCESS ADR(gPowermeters[iIndexPowerMeter]);

	IF NOT PowerMeter.Parameters.xInstalled THEN
		PowerMeter.Alarms := ResetedAlarms;
		RETURN;
	END_IF

	AssignDataComms;

	Alarms;

	//Prepare
	iIndexPowerMeter := iIndexPowerMeter + 1;

END_PROGRAM
```

#### PowerMeter.var - Local variables
```iecst
VAR
	PowerMeter : REFERENCE TO stPowerMeter;
	CommsReset : PowerMeterCommsInputs_typ;
	ModSlaveState : UINT;
	LastError : UINT;
	LastErrorBlockNum : UINT;
	ResetedAlarms : PowerMeterAlarms_typ;
END_VAR
```

### Program Logical/ExtPack/_Extras/SafetyControllerCtrl/SafetyControllerCtrl_v1/SafetyControllerCtrl (IEC)

#### SafetyController.st
```iecst
PROGRAM _CYCLIC

	SafetyController ACCESS ADR(gSafetyController);
	DataFromSafety ACCESS ADR(gReceivedDataModbSafety);

	IF NOT gSafetyController.Parameters.xInstalled THEN
		RETURN;
	END_IF

	AssignDataComms;

	Alarms;

END_PROGRAM
```

### SafetyController.typ
```iecst
TYPE
	SafetyControllerOutputs_typ : 	STRUCT
		xEnablePrinter1 : BOOL; (*OSSD*)
		xEnablePrinter2 : BOOL; (*OSSD*)
		xEnablePrinterBlowers1 : BOOL; (*OSSD*)
		xEnablePrinterBlowers2 : BOOL; (*OSSD*)
		xEnableDryer1 : BOOL; (*OSSD*)
		xEnableDryer2 : BOOL; (*OSSD*)
		xFeederToLine1 : BOOL; (*Relay*)
		xFeederToLine2 : BOOL; (*Relay*)
		xLineToFeeder1 : BOOL; (*Relay*)
		xLineToFeeder2 : BOOL; (*Relay*)
		xPrimerToLine1 : BOOL; (*Relay*)
		xPrimerToLine2 : BOOL; (*Relay*)
		xLineToPrimer1 : BOOL; (*Relay*)
		xLineToPrimer2 : BOOL; (*Relay*)
		xStackerToLine1 : BOOL; (*Relay*)
		xStackerToLine2 : BOOL; (*Relay*)
		xLineToStacker1 : BOOL; (*Relay*)
		xLineToStacker2 : BOOL; (*Relay*)
		xIRToLine1 : BOOL; (*Relay*)
		xIRToLine2 : BOOL; (*Relay*)
		xLineToIR1 : BOOL; (*Relay*)
		xLineToIR2 : BOOL; (*Relay*)
		xUVToLine1 : BOOL; (*Relay*)
		xUVToLine2 : BOOL; (*Relay*)
		xLineToUV1 : BOOL; (*Relay*)
		xLineToUV2 : BOOL; (*Relay*)
		xPrinterToX5 : BOOL; (*Relay*)
	END_STRUCT;
	SafetyControllerInputs_typ : 	STRUCT
		Comms : SafetyControllerCommsInputs_typ;
		xPrinterLightCurtain : BOOL; (*Printer's front side light curtain feedback*)
		xPrinterRearDoorSwitch : BOOL;
		xPrinterFrontDoorSwitch : BOOL;
		xPrinterDoorLock : BOOL; (*Printer's rear side magnetic sensor feedback*)
		xPrinterBacksideEstop : BOOL;
		xPrinterFrontsideEstop : BOOL;
		xPrinterBlowersSwitch : BOOL; (*Switch to cut off blowers drive enables located inside blowers enclusure feedback*)
		xPrinterBlowersEnable : BOOL;
		xPrinterMaintenanceKey : BOOL; (*Maintenance key located in printer's rear side feedback*)
		xDryerBackDoorSwitch1 : BOOL;
		xDryerBackDoorSwitch2 : BOOL;
		xDryerFrontDoorSwitch1 : BOOL;
		xDryerFrontDoorSwitch2 : BOOL;
		xDryerMaintenanceKey : BOOL;
		xIR_SafetyAlarm : BOOL;
		xDryerBlowersEnable : BOOL;
		xDryerBacksideEstop : BOOL;
		xDryerFrontsideEstop : BOOL;
		xFeederEstop : BOOL;
		xPrimerEstop : BOOL;
		xOvervarnishEstop : BOOL;
		xStackerEstop : BOOL;
		xSarmEstop : BOOL;
		xFanDoorSwitch : BOOL;
		xHmiSwitch : BOOL;
		xX5Consent2 : BOOL;
		xX5Consent : BOOL;
	END_STRUCT;
	stSafetyController : 	STRUCT
		Inputs : SafetyControllerInputs_typ;
		Alarms : SafetyControllerAlarms_typ;
		Outputs : SafetyControllerOutputs_typ;
		Status : SafetyControllerStatus_typ;
		Parameters : SafetyParameters_typ;
		Orders : SafetyOrders_typ;
		Commands : SafetyCommands_typ;
	END_STRUCT;
	SafetyControllerCommsInputs_typ : 	STRUCT
		SystemStatus : USINT;
		ExpansionModule : ARRAY[0..15]OF USINT; (*Each expansion module bit is assigned to its input status at that pin*)
		FieldbusInputs : USINT;
		FieldbusProbeStatus : UINT;
		OSSDStatus : UINT;
		DiagnosticCode : UINT;
	END_STRUCT;
	SafetyControllerAlarms_typ : 	STRUCT
		xAlrPrinterEStops : BOOL;
		xAlrPrinter : BOOL;
		xAlrDryer : BOOL;
		xAlrFeeder : BOOL;
		xAlrPrimer : BOOL;
		xAlrOverVarnish : BOOL;
		xAlrStacker : BOOL;
		xAlrSarm : BOOL;
		xCriticalAlarm : BOOL;
		xWarningAlarm : BOOL;
		xAnyAlarm : BOOL;
		xCommsError : BOOL;
		xAlrPrinterLightCurtain : BOOL;
		xAlrBlowersEnclosureSwitchOff : BOOL;
		xAlrPrinterDoorLockKeyActivated : BOOL;
		xAlrPrinterDoorLock : BOOL;
		xAlrPrinterRearDoorSwitch : BOOL;
		xAlrHmiSwitch : BOOL;
		xAlrPrinterFanDoorSwitch : BOOL;
		xAlrPrinterFrontDoorSwitch : BOOL;
		xAlrPrinterFrontEstop : BOOL;
		xAlrPrinterRearEstop : BOOL;
	END_STRUCT;
	SafetyControllerStatus_typ : 	STRUCT
		Version : USINT;
		Comms : SafetyCommsStatus_typ;
		Type : SafetyControllerType_enum;
	END_STRUCT;
	SafetyCommsStatus_typ : 	STRUCT
		xModuleOk : BOOL;
		ModSlaveState : UINT;
		LastError : UINT;
		LastErrorBlockNum : UINT;
		xStopButtonPressed : BOOL;
		ActOverloadError : BOOL;
		ActModbusError : BOOL;
		ActSlvConError : BOOL;
		ActRefreshError : BOOL;
		ActInternalError : BOOL;
		ActConfError : BOOL;
		HistOverloadError : BOOL;
		HistModbusError : BOOL;
		HistSlvConError : BOOL;
		HistRefreshError : BOOL;
		HistInternalError : BOOL;
		HistConfError : BOOL;
		ModbusErrorCnt : UINT;
		ModbusConErrorCnt : UINT;
		ModbusPktRefreshTimeoutCnt : UINT;
		ModbusPktPendPerSec : UINT;
		ModbusMeanResponseTime : UINT;
	END_STRUCT;
	SafetyParameters_typ : 	STRUCT
		xActiveSlaveDiagnosis : BOOL;
		xInstalled : BOOL;
		xSimulationMode : BOOL; (*Defined by the configuration in Automation Studio*)
	END_STRUCT;
	SafetyOrders_typ : 	STRUCT
		xDisableReadBlock : BOOL;
	END_STRUCT;
	SafetyCommands_typ : 	STRUCT
		xReset : BOOL;
	END_STRUCT;
	SafetyControllerType_enum :
		(
		SAFETYCONTROLLERTY_UNDEFINED,
		SAFETYCONTROLLERTY_DEFAULT, (*Default version installed*)
		SAFETYCONTROLLERTY_CUBE_ALPHA, (*Version for Nozomi 2 in Gulliver (first Nz2 manufactured ever) installed*)
		SAFETYCONTROLLERTY_SD, (*Version for display graphics installed*)
		SAFETYCONTROLLERTY_CUBE, (*Version for cube machine model*)
		SAFETYCONTROLLERTY_MECANO, (*Version for Mecano machine model*)
		SAFETYCONTROLLERTY_NOZ2_AQ (*Version for Nozomi 2 water*)
		);
END_TYPE
```

### Program Logical/ExtPack/_Extras/SafetyControllerCtrl/SafetyControllerSim/SafetyControllerSim_v1/SafetyControllerSim (IEC)

#### SafetyControllerSim.st
```iecst
PROGRAM _CYCLIC
	(* Insert code here *)
	SafetyController ACCESS ADR(gSafetyController);
	SimSafetyController ACCESS ADR(gSimSafetyController);

	IF EDGEPOS(SimSafetyController.Commands.xSafetyToDefault) THEN
		SafetyController.Status.Comms.xModuleOk := TRUE;
		//Modules physical inputs
		//Ancillaries
		SimSafetyController.Inputs.xFeederEstop				:= TRUE;
		SimSafetyController.Inputs.xPrimerEstop 			:= TRUE;
		SimSafetyController.Inputs.xOvervarnishEstop 		:= TRUE;
		SimSafetyController.Inputs.xStackerEstop 			:= TRUE;
		SimSafetyController.Inputs.xSarmEstop				:= TRUE;

		//Dryer
		SimSafetyController.Inputs.xDryerBacksideEstop 		:= TRUE;
		SimSafetyController.Inputs.xDryerFrontsideEstop 	:= TRUE;
		SimSafetyController.Inputs.xDryerFrontDoorSwitch1	:= TRUE;
		SimSafetyController.Inputs.xDryerFrontDoorSwitch2	:= TRUE;
		SimSafetyController.Inputs.xDryerBackDoorSwitch1	:= TRUE;
		SimSafetyController.Inputs.xDryerBackDoorSwitch2	:= TRUE;
		SimSafetyController.Inputs.xDryerMaintenanceKey		:= FALSE;
		SimSafetyController.Inputs.xDryerBlowersEnable		:= TRUE;

		//Printer
		SimSafetyController.Inputs.xPrinterMaintenanceKey 	:= FALSE;
		SimSafetyController.Inputs.xPrinterBlowersEnable	:= TRUE;
		SimSafetyController.Inputs.xPrinterBlowersSwitch	:= TRUE;
		SimSafetyController.Inputs.xPrinterLightCurtain 	:= TRUE;
		SimSafetyController.Inputs.xPrinterDoorLock 		:= TRUE;
		SimSafetyController.Inputs.xPrinterBacksideEstop 	:= TRUE;
		SimSafetyController.Inputs.xPrinterFrontsideEstop 	:= TRUE;

		//OSSD Outputs
		SimSafetyController.Outputs.xEnablePrinter1 		:= TRUE;
		SimSafetyController.Outputs.xEnablePrinterBlowers1 	:= TRUE;
		SimSafetyController.Outputs.xEnableDryer1			:= TRUE;

		SafetyController.Status.Comms.xModuleOk 			:= TRUE;

		//Fieldbus probe
		//Inputs
		SimSafetyController.Inputs.xPrinterRearDoorSwitch 	:= TRUE;
		SimSafetyController.Inputs.xHmiSwitch 				:= TRUE;
		SimSafetyController.Inputs.xPrinterFrontDoorSwitch 	:= TRUE;
		SimSafetyController.Inputs.xX5Consent 				:= TRUE;
		SimSafetyController.Inputs.xFanDoorSwitch	 		:= TRUE;

		//Outputs
		SimSafetyController.Outputs.xEnablePrinter1 		:= TRUE;
		SimSafetyController.Outputs.xPrinterToX5 			:= TRUE;

		//Resetting command
		SimSafetyController.Commands.xSafetyToDefault		:= FALSE;
	END_IF

	SafetyController.Inputs := SimSafetyController.Inputs;

END_PROGRAM
```

### Package Logical/ExtPack/InksCtrl - Inks Control Logic package

### Package Logical/ExtPack/InksCtrl/InksCtrl_v3 - Inks control logic package

### Program Logical/ExtPack/InksCtrl/InksCtrl_v3/InksCtrl (IEC) - Inks Control Program

#### Constants.var
```iecst
VAR CONSTANT
	lc_rHighPresEnterStable : REAL := 14.0;
	lc_rHighPresExitStable : REAL := 15.0;
	lc_rLowPresEnterStable : REAL := 2.0;
	lc_rLowPresExitStable : REAL := 0.0;
	lc_rCyclePwm : REAL := 2.0; (*Time in seconds of the Cycle for the temp control*)
	Ic_rMinDiffMinMaxCtrlVoltage : REAL := 0.5; (*for the conversion to the slope in the graph V-%DC.	*)
	LC_MAX_MENISCUS_TO_STARTED : INT := 50; (*MAx diff between meniscus and meniscus measured for changing filling pump PID while is starting*) (*gc_rSetPointBNegativeMode8 : REAL := 25.0;*)
	LC_MIN_MENISCUS_TO_STARTED : INT := 0; (*Min diff between meniscus and meniscus measured for changing filling pump PID while is starting*)
	lc_tiTimeStoppingPsu : TIME := T#3S;
	lc_rDiffBetweenPumpsDCLimit : REAL := 84.0;
	MAX_DIFFCTRLTEMP_ALR : REAL := 2.5; (* Limit to define Error in Control temperature with the output signal. AlarmStop. Value in C degree*)
	MAX_DIFFCTRLTEMP_WRNG : REAL := 1.0; (* Limit to define Error in Control temperature. Value in C degree*)
	SETPOINT_MENISCUS_DRIP : REAL := -20.0; (*Sp Meniscus for dripping*)
	MAX_DIFFCTRLTEMPHIGH_ALR : REAL := 4; (* Limit to define Error in Control temperature with the heater resistance. AlarmStop. Value in C degree*)
END_VAR
```
